LIN {X 0,Y 298.919,Z 282.875,A -85,B 0,C 180,E1 -16201.349,E2 -16201.349} C_VEL
LIN {X 0,Y 298.794,Z 282.889,A -85,B 0,C 180,E1 -16206.755,E2 -16206.755} C_VEL
LIN {X 0,Y 298.677,Z 282.907,A -85,B 0,C 180,E1 -16209.482,E2 -16209.482} C_VEL
LIN {X 0,Y 298.549,Z 282.919,A -85,B 0,C 180,E1 -16213.617,E2 -16213.617} C_VEL
LIN {X 0,Y 298.546,Z 282.921,A -85,B 0,C 180,E1 -16216.41,E2 -16216.41} C_VEL
LIN {X 0,Y 298.509,Z 282.922,A -85,B 0,C 180,E1 -16219.656,E2 -16219.656} C_VEL
LIN {X 0,Y 298.48,Z 283.099,A -85,B 0,C 180,E1 -16223.325,E2 -16223.325} C_VEL
LIN {X 0,Y 298.814,Z 284.83,A -85,B 0,C 180,E1 -16226.655,E2 -16226.655} C_VEL
LIN {X 0,Y 299.125,Z 286.68,A -85,B 0,C 180,E1 -16229.622,E2 -16229.622} C_VEL
LIN {X 0,Y 299.687,Z 290.164,A -85,B 0,C 180,E1 -16234.253,E2 -16234.253} C_VEL
LIN {X 0,Y 300.171,Z 292.989,A -85,B 0,C 180,E1 -16237.5,E2 -16237.5} C_VEL
LIN {X 0,Y 300.838,Z 297.077,A -85,B 0,C 180,E1 -16241.622,E2 -16241.622} C_VEL
LIN {X 0,Y 301.665,Z 301.596,A -85,B 0,C 180,E1 -16245.661,E2 -16245.661} C_VEL
LIN {X 0,Y 301.692,Z 304.757,A -85,B 0,C 180,E1 -16248.199,E2 -16248.199} C_VEL
LIN {X 0,Y 300.821,Z 309.639,A -85,B 0,C 180,E1 -16251.75,E2 -16251.75} C_VEL
LIN {X 0,Y 300.436,Z 312.082,A -85,B 0,C 180,E1 -16253.389,E2 -16253.389} C_VEL
LIN {X 0,Y 301.353,Z 315.27,A -85,B 0,C 180,E1 -16253.65,E2 -16253.65} C_VEL
LIN {X 0,Y 302.505,Z 317.919,A -85,B 0,C 180,E1 -16253.94,E2 -16253.94} C_VEL
LIN {X 0,Y 307.209,Z 331.176,A -85,B 0,C 180,E1 -16255.276,E2 -16255.276} C_VEL
LIN {X 0,Y 310.679,Z 343.941,A -85,B 0,C 180,E1 -16256.565,E2 -16256.565} C_VEL
LIN {X 0,Y 312.999,Z 356.009,A -85,B 0,C 180,E1 -16257.802,E2 -16257.802} C_VEL
LIN {X 0,Y 314.515,Z 369.598,A -85,B 0,C 180,E1 -16259.261,E2 -16259.261} C_VEL
LIN {X 0,Y 315.116,Z 381.128,A -85,B 0,C 180,E1 -16260.617,E2 -16260.617} C_VEL
LIN {X 0,Y 312.318,Z 395,A -85,B 0,C 180,E1 -16262.166,E2 -16262.166} C_VEL
LIN {X 0,Y 309.669,Z 406.556,A -85,B 0,C 180,E1 -16263.734,E2 -16263.734} C_VEL
LIN {X 0,Y 306.844,Z 418.279,A -85,B 0,C 180,E1 -16265.653,E2 -16265.653} C_VEL
LIN {X 0,Y 304.314,Z 429.043,A -85,B 0,C 180,E1 -16267.799,E2 -16267.799} C_VEL
LIN {X 0,Y 302.202,Z 438.027,A -85,B 0,C 180,E1 -16269.94,E2 -16269.94} C_VEL
LIN {X 0,Y 300.309,Z 446.263,A -85,B 0,C 180,E1 -16272.289,E2 -16272.289} C_VEL
LIN {X 0,Y 298.594,Z 453.992,A -85,B 0,C 180,E1 -16274.996,E2 -16274.996} C_VEL
LIN {X 0,Y 297.601,Z 460.201,A -85,B 0,C 180,E1 -16277.73,E2 -16277.73} C_VEL
LIN {X 0,Y 296.971,Z 465.011,A -85,B 0,C 180,E1 -16280.465,E2 -16280.465} C_VEL
LIN {X 0,Y 296.728,Z 468.523,A -85,B 0,C 180,E1 -16283.2,E2 -16283.2} C_VEL
LIN {X 0,Y 296.652,Z 470.817,A -85,B 0,C 180,E1 -16285.925,E2 -16285.925} C_VEL
LIN {X 0,Y 296.663,Z 471.931,A -85,B 0,C 180,E1 -16288.643,E2 -16288.643} C_VEL
LIN {X 0,Y 296.733,Z 472.054,A -85,B 0,C 180,E1 -16290.001,E2 -16290.001} C_VEL
LIN {X 0,Y 296.633,Z 471.4,A -85,B 0,C 180,E1 -16292.717,E2 -16292.717} C_VEL
LIN {X 0,Y 296.692,Z 469.509,A -85,B 0,C 180,E1 -16295.438,E2 -16295.438} C_VEL
LIN {X 0,Y 296.827,Z 466.384,A -85,B 0,C 180,E1 -16298.168,E2 -16298.168} C_VEL
LIN {X 0,Y 297.197,Z 461.97,A -85,B 0,C 180,E1 -16300.906,E2 -16300.906} C_VEL
LIN {X 0,Y 298.046,Z 456.167,A -85,B 0,C 180,E1 -16303.64,E2 -16303.64} C_VEL
LIN {X 0,Y 299.38,Z 448.82,A -85,B 0,C 180,E1 -16306.363,E2 -16306.363} C_VEL
LIN {X 0,Y 300.944,Z 440.958,A -85,B 0,C 180,E1 -16308.731,E2 -16308.731} C_VEL
LIN {X 0,Y 303.074,Z 431.526,A -85,B 0,C 180,E1 -16311.066,E2 -16311.066} C_VEL
LIN {X 0,Y 305.057,Z 421.918,A -85,B 0,C 180,E1 -16313.058,E2 -16313.058} C_VEL
LIN {X 0,Y 307.558,Z 410.541,A -85,B 0,C 180,E1 -16315.009,E2 -16315.009} C_VEL
LIN {X 0,Y 310.005,Z 398.045,A -85,B 0,C 180,E1 -16316.782,E2 -16316.782} C_VEL
LIN {X 0,Y 312.757,Z 384.378,A -85,B 0,C 180,E1 -16318.333,E2 -16318.333} C_VEL
LIN {X 0,Y 313.53,Z 379.839,A -85,B 0,C 180,E1 -16318.782,E2 -16318.782} C_VEL
LIN {X 0,Y 311.965,Z 365.595,A -85,B 0,C 180,E1 -16320.332,E2 -16320.332} C_VEL
LIN {X 0,Y 309.68,Z 351.608,A -85,B 0,C 180,E1 -16321.673,E2 -16321.673} C_VEL
LIN {X 0,Y 306.111,Z 335.839,A -85,B 0,C 180,E1 -16323.017,E2 -16323.017} C_VEL
LIN {X 0,Y 301.772,Z 321.161,A -85,B 0,C 180,E1 -16324.129,E2 -16324.129} C_VEL
LIN {X 0,Y 300.006,Z 315.466,A -85,B 0,C 180,E1 -16324.519,E2 -16324.519} C_VEL
LIN {X 0,Y 299.925,Z 314.804,A -85,B 0,C 180,E1 -16324.578,E2 -16324.578} C_VEL
LIN {X 0,Y 300.788,Z 309.235,A -85,B 0,C 180,E1 -16328.257,E2 -16328.257} C_VEL
LIN {X 0,Y 301.384,Z 305.562,A -85,B 0,C 180,E1 -16330.764,E2 -16330.764} C_VEL
LIN {X 0,Y 301.617,Z 303.07,A -85,B 0,C 180,E1 -16332.512,E2 -16332.512} C_VEL
LIN {X 0,Y 301.57,Z 300.589,A -85,B 0,C 180,E1 -16334.359,E2 -16334.359} C_VEL
LIN {X 0,Y 300.579,Z 295.456,A -85,B 0,C 180,E1 -16338.437,E2 -16338.437} C_VEL
LIN {X 0,Y 299.661,Z 290.232,A -85,B 0,C 180,E1 -16342.884,E2 -16342.884} C_VEL
LIN {X 0,Y 299.197,Z 287.18,A -85,B 0,C 180,E1 -16345.683,E2 -16345.683} C_VEL
LIN {X 0,Y 298.44,Z 283.034,A -85,B 0,C 180,E1 -16349.776,E2 -16349.776} C_VEL
LIN {X 0,Y 298.484,Z 282.93,A -85,B 0,C 180,E1 -16353.476,E2 -16353.476} C_VEL
LIN {X 0,Y 298.442,Z 282.937,A -85,B 0,C 180,E1 -16356.697,E2 -16356.697} C_VEL
LIN {X 0,Y 298.546,Z 282.923,A -85,B 0,C 180,E1 -16360.756,E2 -16360.756} C_VEL
LIN {X 0,Y 298.6,Z 282.916,A -85,B 0,C 180,E1 -16364.994,E2 -16364.994} C_VEL
LIN {X 0,Y 298.597,Z 282.915,A -85,B 0,C 180,E1 -16369.145,E2 -16369.145} C_VEL
LIN {X 0,Y 298.718,Z 282.9,A -85,B 0,C 180,E1 -16371.883,E2 -16371.883} C_VEL
LIN {X 0,Y 298.648,Z 282.911,A -85,B 0,C 180,E1 -16374.597,E2 -16374.597} C_VEL
LIN {X 0,Y 298.928,Z 282.875,A -85,B 0,C 180,E1 -16378.651,E2 -16378.651} C_VEL
LIN {X 0,Y 298.928,Z 282.871,A -85,B 0,C 180,E1 -16381.346,E2 -16381.346} C_VEL
LIN {X 0,Y 298.801,Z 282.889,A -85,B 0,C 180,E1 -16386.752,E2 -16386.752} C_VEL
LIN {X 0,Y 298.684,Z 282.902,A -85,B 0,C 180,E1 -16389.479,E2 -16389.479} C_VEL
LIN {X 0,Y 298.554,Z 282.914,A -85,B 0,C 180,E1 -16393.614,E2 -16393.614} C_VEL
LIN {X 0,Y 298.551,Z 282.921,A -85,B 0,C 180,E1 -16396.407,E2 -16396.407} C_VEL
LIN {X 0,Y 298.513,Z 282.92,A -85,B 0,C 180,E1 -16399.653,E2 -16399.653} C_VEL
LIN {X 0,Y 298.458,Z 282.931,A -85,B 0,C 180,E1 -16403.596,E2 -16403.596} C_VEL
LIN {X 0,Y 298.486,Z 282.924,A -85,B 0,C 180,E1 -16406.573,E2 -16406.573} C_VEL
LIN {X 0,Y 298.416,Z 282.933,A -85,B 0,C 180,E1 -16409.639,E2 -16409.639} C_VEL
LIN {X 0,Y 298.394,Z 282.938,A -85,B 0,C 180,E1 -16412.798,E2 -16412.798} C_VEL
LIN {X 0,Y 298.462,Z 282.926,A -85,B 0,C 180,E1 -16416.81,E2 -16416.81} C_VEL
LIN {X 0,Y 298.411,Z 282.936,A -85,B 0,C 180,E1 -16421.255,E2 -16421.255} C_VEL
LIN {X 0,Y 298.413,Z 282.935,A -85,B 0,C 180,E1 -16425.045,E2 -16425.045} C_VEL
LIN {X 0,Y 298.45,Z 282.927,A -85,B 0,C 180,E1 -16428.748,E2 -16428.748} C_VEL
LIN {X 0,Y 298.442,Z 282.934,A -85,B 0,C 180,E1 -16432.245,E2 -16432.245} C_VEL
LIN {X 0,Y 298.402,Z 282.937,A -85,B 0,C 180,E1 -16435.579,E2 -16435.579} C_VEL
LIN {X 0,Y 298.389,Z 282.94,A -85,B 0,C 180,E1 -16438.79,E2 -16438.79} C_VEL
LIN {X 0,Y 298.469,Z 282.934,A -85,B 0,C 180,E1 -16441.904,E2 -16441.904} C_VEL
LIN {X 0,Y 298.478,Z 282.927,A -85,B 0,C 180,E1 -16444.922,E2 -16444.922} C_VEL
LIN {X 0,Y 298.442,Z 282.934,A -85,B 0,C 180,E1 -16449.314,E2 -16449.314} C_VEL
LIN {X 0,Y 298.529,Z 282.92,A -85,B 0,C 180,E1 -16452.178,E2 -16452.178} C_VEL
LIN {X 0,Y 298.584,Z 282.917,A -85,B 0,C 180,E1 -16454.993,E2 -16454.993} C_VEL
LIN {X 0,Y 298.586,Z 282.916,A -85,B 0,C 180,E1 -16459.145,E2 -16459.145} C_VEL
LIN {X 0,Y 298.748,Z 282.888,A -85,B 0,C 180,E1 -16461.885,E2 -16461.885} C_VEL
LIN {X 0,Y 298.592,Z 282.915,A -85,B 0,C 180,E1 -16464.597,E2 -16464.597} C_VEL
LIN {X 0,Y 298.28,Z 282.958,A -85,B 0,C 180,E1 -16467.298,E2 -16467.298} C_VEL
LIN {X 0,Y 298.703,Z 283.826,A -85,B 0,C 180,E1 -16468.689,E2 -16468.689} C_VEL
LIN {X 0,Y 299.818,Z 287.044,A -85,B 0,C 180,E1 -16468.935,E2 -16468.935} C_VEL
LIN {X 0,Y 305.646,Z 301.861,A -85,B 0,C 180,E1 -16470.26,E2 -16470.26} C_VEL
LIN {X 0,Y 310.151,Z 313.487,A -85,B 0,C 180,E1 -16471.449,E2 -16471.449} C_VEL
LIN {X 0,Y 314.135,Z 327.182,A -85,B 0,C 180,E1 -16472.928,E2 -16472.928} C_VEL
LIN {X 0,Y 315.72,Z 333.801,A -85,B 0,C 180,E1 -16473.69,E2 -16473.69} C_VEL
LIN {X 0,Y 315.258,Z 338.882,A -85,B 0,C 180,E1 -16474.154,E2 -16474.154} C_VEL
LIN {X 0,Y 313.237,Z 352.066,A -85,B 0,C 180,E1 -16475.471,E2 -16475.471} C_VEL
LIN {X 0,Y 311.014,Z 364.333,A -85,B 0,C 180,E1 -16476.958,E2 -16476.958} C_VEL
LIN {X 0,Y 308.798,Z 375.976,A -85,B 0,C 180,E1 -16478.671,E2 -16478.671} C_VEL
LIN {X 0,Y 306.535,Z 386.753,A -85,B 0,C 180,E1 -16480.568,E2 -16480.568} C_VEL
LIN {X 0,Y 304.365,Z 396.697,A -85,B 0,C 180,E1 -16482.671,E2 -16482.671} C_VEL
LIN {X 0,Y 302.151,Z 406.39,A -85,B 0,C 180,E1 -16485.168,E2 -16485.168} C_VEL
LIN {X 0,Y 300.48,Z 414.358,A -85,B 0,C 180,E1 -16487.701,E2 -16487.701} C_VEL
LIN {X 0,Y 299.164,Z 420.286,A -85,B 0,C 180,E1 -16490.008,E2 -16490.008} C_VEL
LIN {X 0,Y 298.31,Z 424.761,A -85,B 0,C 180,E1 -16492.144,E2 -16492.144} C_VEL
LIN {X 0,Y 297.623,Z 428.608,A -85,B 0,C 180,E1 -16494.407,E2 -16494.407} C_VEL
LIN {X 0,Y 297.086,Z 431.545,A -85,B 0,C 180,E1 -16496.709,E2 -16496.709} C_VEL
LIN {X 0,Y 296.755,Z 433.529,A -85,B 0,C 180,E1 -16498.809,E2 -16498.809} C_VEL
LIN {X 0,Y 296.592,Z 434.977,A -85,B 0,C 180,E1 -16501.459,E2 -16501.459} C_VEL
LIN {X 0,Y 296.562,Z 435.382,A -85,B 0,C 180,E1 -16503.963,E2 -16503.963} C_VEL
LIN {X 0,Y 296.697,Z 434.896,A -85,B 0,C 180,E1 -16506.357,E2 -16506.357} C_VEL
LIN {X 0,Y 297.054,Z 433.533,A -85,B 0,C 180,E1 -16508.674,E2 -16508.674} C_VEL
LIN {X 0,Y 297.695,Z 430.916,A -85,B 0,C 180,E1 -16511.377,E2 -16511.377} C_VEL
LIN {X 0,Y 298.593,Z 427.274,A -85,B 0,C 180,E1 -16513.973,E2 -16513.973} C_VEL
LIN {X 0,Y 299.829,Z 422.32,A -85,B 0,C 180,E1 -16516.604,E2 -16516.604} C_VEL
LIN {X 0,Y 301.488,Z 415.919,A -85,B 0,C 180,E1 -16519.256,E2 -16519.256} C_VEL
LIN {X 0,Y 303.672,Z 407.901,A -85,B 0,C 180,E1 -16521.893,E2 -16521.893} C_VEL
LIN {X 0,Y 305.787,Z 399.629,A -85,B 0,C 180,E1 -16524.11,E2 -16524.11} C_VEL
LIN {X 0,Y 308.375,Z 389.763,A -85,B 0,C 180,E1 -16526.288,E2 -16526.288} C_VEL
LIN {X 0,Y 310.943,Z 379.241,A -85,B 0,C 180,E1 -16528.217,E2 -16528.217} C_VEL
LIN {X 0,Y 313.577,Z 367.883,A -85,B 0,C 180,E1 -16529.94,E2 -16529.94} C_VEL
LIN {X 0,Y 316.01,Z 355.888,A -85,B 0,C 180,E1 -16531.456,E2 -16531.456} C_VEL
LIN {X 0,Y 318.371,Z 343.09,A -85,B 0,C 180,E1 -16532.775,E2 -16532.775} C_VEL
LIN {X 0,Y 319.093,Z 338.798,A -85,B 0,C 180,E1 -16533.161,E2 -16533.161} C_VEL
LIN {X 0,Y 316.264,Z 327.369,A -85,B 0,C 180,E1 -16534.642,E2 -16534.642} C_VEL
LIN {X 0,Y 311.737,Z 314.131,A -85,B 0,C 180,E1 -16536.338,E2 -16536.338} C_VEL
LIN {X 0,Y 306.157,Z 301.839,A -85,B 0,C 180,E1 -16537.966,E2 -16537.966} C_VEL
LIN {X 0,Y 302.671,Z 295.179,A -85,B 0,C 180,E1 -16538.863,E2 -16538.863} C_VEL
LIN {X 0,Y 300.761,Z 291.735,A -85,B 0,C 180,E1 -16539.323,E2 -16539.323} C_VEL
LIN {X 0,Y 299.162,Z 288.982,A -85,B 0,C 180,E1 -16539.713,E2 -16539.713} C_VEL
LIN {X 0,Y 298.817,Z 287.666,A -85,B 0,C 180,E1 -16539.845,E2 -16539.845} C_VEL
LIN {X 0,Y 298.868,Z 287.057,A -85,B 0,C 180,E1 -16541.023,E2 -16541.023} C_VEL
LIN {X 0,Y 298.189,Z 286.627,A -85,B 0,C 180,E1 -16542.146,E2 -16542.146} C_VEL
LIN {X 0,Y 295.347,Z 286.279,A -85,B 0,C 180,E1 -16543.98,E2 -16543.98} C_VEL
LIN {X 0,Y 292.934,Z 286.066,A -85,B 0,C 180,E1 -16545.468,E2 -16545.468} C_VEL
LIN {X 0,Y 291.882,Z 285.781,A -85,B 0,C 180,E1 -16546.62,E2 -16546.62} C_VEL
LIN {X 0,Y 291.786,Z 285.628,A -85,B 0,C 180,E1 -16547.009,E2 -16547.009} C_VEL
LIN {X 0,Y 291.735,Z 283.882,A -85,B 0,C 180,E1 -16551.691,E2 -16551.691} C_VEL
LIN {X 0,Y 291.627,Z 283.783,A -85,B 0,C 180,E1 -16554.47,E2 -16554.47} C_VEL
LIN {X 0,Y 291.885,Z 283.752,A -85,B 0,C 180,E1 -16558.622,E2 -16558.622} C_VEL
LIN {X 0,Y 291.886,Z 283.75,A -85,B 0,C 180,E1 -16561.381,E2 -16561.381} C_VEL
LIN {X 0,Y 291.743,Z 283.768,A -85,B 0,C 180,E1 -16566.919,E2 -16566.919} C_VEL
LIN {X 0,Y 291.626,Z 283.785,A -85,B 0,C 180,E1 -16569.713,E2 -16569.713} C_VEL
LIN {X 0,Y 291.519,Z 283.797,A -85,B 0,C 180,E1 -16573.952,E2 -16573.952} C_VEL
LIN {X 0,Y 291.484,Z 283.797,A -85,B 0,C 180,E1 -16576.819,E2 -16576.819} C_VEL
LIN {X 0,Y 291.448,Z 283.803,A -85,B 0,C 180,E1 -16579.876,E2 -16579.876} C_VEL
LIN {X 0,Y 291.396,Z 283.873,A -85,B 0,C 180,E1 -16581.211,E2 -16581.211} C_VEL
LIN {X 0,Y 291.623,Z 285.187,A -85,B 0,C 180,E1 -16584.187,E2 -16584.187} C_VEL
LIN {X 0,Y 291.966,Z 286.805,A -85,B 0,C 180,E1 -16587.218,E2 -16587.218} C_VEL
LIN {X 0,Y 292.243,Z 288.784,A -85,B 0,C 180,E1 -16590.334,E2 -16590.334} C_VEL
LIN {X 0,Y 292.62,Z 291.137,A -85,B 0,C 180,E1 -16593.533,E2 -16593.533} C_VEL
LIN {X 0,Y 293.13,Z 293.884,A -85,B 0,C 180,E1 -16596.828,E2 -16596.828} C_VEL
LIN {X 0,Y 293.626,Z 297.12,A -85,B 0,C 180,E1 -16600.261,E2 -16600.261} C_VEL
LIN {X 0,Y 294.415,Z 301.316,A -85,B 0,C 180,E1 -16604.265,E2 -16604.265} C_VEL
LIN {X 0,Y 294.753,Z 303.579,A -85,B 0,C 180,E1 -16606.255,E2 -16606.255} C_VEL
LIN {X 0,Y 294.711,Z 305.868,A -85,B 0,C 180,E1 -16608.11,E2 -16608.11} C_VEL
LIN {X 0,Y 293.689,Z 311.336,A -85,B 0,C 180,E1 -16612.185,E2 -16612.185} C_VEL
LIN {X 0,Y 294.665,Z 314.757,A -85,B 0,C 180,E1 -16612.509,E2 -16612.509} C_VEL
LIN {X 0,Y 295.761,Z 317.224,A -85,B 0,C 180,E1 -16612.804,E2 -16612.804} C_VEL
LIN {X 0,Y 300.269,Z 329.416,A -85,B 0,C 180,E1 -16614.128,E2 -16614.128} C_VEL
LIN {X 0,Y 304.198,Z 343.339,A -85,B 0,C 180,E1 -16615.627,E2 -16615.627} C_VEL
LIN {X 0,Y 306.889,Z 357.513,A -85,B 0,C 180,E1 -16617.159,E2 -16617.159} C_VEL
LIN {X 0,Y 308.218,Z 370.175,A -85,B 0,C 180,E1 -16618.584,E2 -16618.584} C_VEL
LIN {X 0,Y 308.727,Z 382.548,A -85,B 0,C 180,E1 -16620.097,E2 -16620.097} C_VEL
LIN {X 0,Y 305.76,Z 396.324,A -85,B 0,C 180,E1 -16621.702,E2 -16621.702} C_VEL
LIN {X 0,Y 302.793,Z 408.654,A -85,B 0,C 180,E1 -16623.462,E2 -16623.462} C_VEL
LIN {X 0,Y 299.919,Z 419.961,A -85,B 0,C 180,E1 -16625.423,E2 -16625.423} C_VEL
LIN {X 0,Y 297.23,Z 431.049,A -85,B 0,C 180,E1 -16627.771,E2 -16627.771} C_VEL
LIN {X 0,Y 294.831,Z 440.289,A -85,B 0,C 180,E1 -16630.144,E2 -16630.144} C_VEL
LIN {X 0,Y 293.012,Z 448.031,A -85,B 0,C 180,E1 -16632.554,E2 -16632.554} C_VEL
LIN {X 0,Y 291.352,Z 455.328,A -85,B 0,C 180,E1 -16635.329,E2 -16635.329} C_VEL
LIN {X 0,Y 290.374,Z 461.138,A -85,B 0,C 180,E1 -16638.129,E2 -16638.129} C_VEL
LIN {X 0,Y 289.911,Z 464.645,A -85,B 0,C 180,E1 -16640.231,E2 -16640.231} C_VEL
LIN {X 0,Y 289.649,Z 468.132,A -85,B 0,C 180,E1 -16643.033,E2 -16643.033} C_VEL
LIN {X 0,Y 289.57,Z 470.402,A -85,B 0,C 180,E1 -16645.825,E2 -16645.825} C_VEL
LIN {X 0,Y 289.575,Z 471.496,A -85,B 0,C 180,E1 -16648.61,E2 -16648.61} C_VEL
LIN {X 0,Y 289.646,Z 471.609,A -85,B 0,C 180,E1 -16650.001,E2 -16650.001} C_VEL
LIN {X 0,Y 289.558,Z 470.938,A -85,B 0,C 180,E1 -16652.783,E2 -16652.783} C_VEL
LIN {X 0,Y 289.642,Z 468.827,A -85,B 0,C 180,E1 -16655.814,E2 -16655.814} C_VEL
LIN {X 0,Y 289.837,Z 464.915,A -85,B 0,C 180,E1 -16659.069,E2 -16659.069} C_VEL
LIN {X 0,Y 290.376,Z 460.158,A -85,B 0,C 180,E1 -16661.873,E2 -16661.873} C_VEL
LIN {X 0,Y 291.365,Z 453.952,A -85,B 0,C 180,E1 -16664.672,E2 -16664.672} C_VEL
LIN {X 0,Y 292.919,Z 446.146,A -85,B 0,C 180,E1 -16667.453,E2 -16667.453} C_VEL
LIN {X 0,Y 294.737,Z 437.817,A -85,B 0,C 180,E1 -16669.865,E2 -16669.865} C_VEL
LIN {X 0,Y 297.028,Z 427.814,A -85,B 0,C 180,E1 -16672.247,E2 -16672.247} C_VEL
LIN {X 0,Y 299.237,Z 417.559,A -85,B 0,C 180,E1 -16674.269,E2 -16674.269} C_VEL
LIN {X 0,Y 301.992,Z 405.418,A -85,B 0,C 180,E1 -16676.243,E2 -16676.243} C_VEL
LIN {X 0,Y 304.194,Z 394.565,A -85,B 0,C 180,E1 -16677.709,E2 -16677.709} C_VEL
LIN {X 0,Y 306.655,Z 382.432,A -85,B 0,C 180,E1 -16679.063,E2 -16679.063} C_VEL
LIN {X 0,Y 306.745,Z 378.889,A -85,B 0,C 180,E1 -16679.465,E2 -16679.465} C_VEL
LIN {X 0,Y 305.283,Z 365.72,A -85,B 0,C 180,E1 -16680.941,E2 -16680.941} C_VEL
LIN {X 0,Y 303.087,Z 352,A -85,B 0,C 180,E1 -16682.307,E2 -16682.307} C_VEL
LIN {X 0,Y 299.567,Z 336.367,A -85,B 0,C 180,E1 -16683.689,E2 -16683.689} C_VEL
LIN {X 0,Y 294.917,Z 320.751,A -85,B 0,C 180,E1 -16684.933,E2 -16684.933} C_VEL
LIN {X 0,Y 293.131,Z 315.095,A -85,B 0,C 180,E1 -16685.343,E2 -16685.343} C_VEL
LIN {X 0,Y 293.075,Z 314.35,A -85,B 0,C 180,E1 -16685.404,E2 -16685.404} C_VEL
LIN {X 0,Y 294.007,Z 308.671,A -85,B 0,C 180,E1 -16689.297,E2 -16689.297} C_VEL
LIN {X 0,Y 294.587,Z 304.45,A -85,B 0,C 180,E1 -16692.304,E2 -16692.304} C_VEL
LIN {X 0,Y 294.564,Z 301.822,A -85,B 0,C 180,E1 -16694.292,E2 -16694.292} C_VEL
LIN {X 0,Y 293.684,Z 297.304,A -85,B 0,C 180,E1 -16697.927,E2 -16697.927} C_VEL
LIN {X 0,Y 292.948,Z 293.24,A -85,B 0,C 180,E1 -16701.408,E2 -16701.408} C_VEL
LIN {X 0,Y 292.364,Z 289.487,A -85,B 0,C 180,E1 -16704.818,E2 -16704.818} C_VEL
LIN {X 0,Y 291.818,Z 286.231,A -85,B 0,C 180,E1 -16708.004,E2 -16708.004} C_VEL
LIN {X 0,Y 291.404,Z 283.813,A -85,B 0,C 180,E1 -16710.704,E2 -16710.704} C_VEL
LIN {X 0,Y 291.419,Z 283.811,A -85,B 0,C 180,E1 -16714.271,E2 -16714.271} C_VEL
LIN {X 0,Y 291.388,Z 283.814,A -85,B 0,C 180,E1 -16717.299,E2 -16717.299} C_VEL
LIN {X 0,Y 291.464,Z 283.805,A -85,B 0,C 180,E1 -16720.269,E2 -16720.269} C_VEL
LIN {X 0,Y 291.561,Z 283.795,A -85,B 0,C 180,E1 -16724.623,E2 -16724.623} C_VEL
LIN {X 0,Y 291.541,Z 283.796,A -85,B 0,C 180,E1 -16728.879,E2 -16728.879} C_VEL
LIN {X 0,Y 291.669,Z 283.778,A -85,B 0,C 180,E1 -16731.686,E2 -16731.686} C_VEL
LIN {X 0,Y 291.617,Z 283.788,A -85,B 0,C 180,E1 -16734.467,E2 -16734.467} C_VEL
LIN {X 0,Y 291.894,Z 283.752,A -85,B 0,C 180,E1 -16738.619,E2 -16738.619} C_VEL
LIN {X 0,Y 291.894,Z 283.748,A -85,B 0,C 180,E1 -16741.378,E2 -16741.378} C_VEL
LIN {X 0,Y 291.75,Z 283.766,A -85,B 0,C 180,E1 -16746.916,E2 -16746.916} C_VEL
LIN {X 0,Y 291.633,Z 283.781,A -85,B 0,C 180,E1 -16749.71,E2 -16749.71} C_VEL
LIN {X 0,Y 291.524,Z 283.791,A -85,B 0,C 180,E1 -16753.948,E2 -16753.948} C_VEL
LIN {X 0,Y 291.489,Z 283.798,A -85,B 0,C 180,E1 -16756.816,E2 -16756.816} C_VEL
LIN {X 0,Y 291.452,Z 283.799,A -85,B 0,C 180,E1 -16759.873,E2 -16759.873} C_VEL
LIN {X 0,Y 291.401,Z 283.813,A -85,B 0,C 180,E1 -16764.203,E2 -16764.203} C_VEL
LIN {X 0,Y 291.419,Z 283.803,A -85,B 0,C 180,E1 -16767.27,E2 -16767.27} C_VEL
LIN {X 0,Y 291.333,Z 283.819,A -85,B 0,C 180,E1 -16770.435,E2 -16770.435} C_VEL
LIN {X 0,Y 291.343,Z 283.819,A -85,B 0,C 180,E1 -16773.696,E2 -16773.696} C_VEL
LIN {X 0,Y 291.391,Z 283.807,A -85,B 0,C 180,E1 -16777.256,E2 -16777.256} C_VEL
LIN {X 0,Y 291.368,Z 283.813,A -85,B 0,C 180,E1 -16780.634,E2 -16780.634} C_VEL
LIN {X 0,Y 291.339,Z 283.817,A -85,B 0,C 180,E1 -16784.39,E2 -16784.39} C_VEL
LIN {X 0,Y 291.384,Z 283.808,A -85,B 0,C 180,E1 -16788.388,E2 -16788.388} C_VEL
LIN {X 0,Y 291.383,Z 283.811,A -85,B 0,C 180,E1 -16791.162,E2 -16791.162} C_VEL
LIN {X 0,Y 291.38,Z 283.808,A -85,B 0,C 180,E1 -16794.628,E2 -16794.628} C_VEL
LIN {X 0,Y 291.366,Z 283.817,A -85,B 0,C 180,E1 -16797.949,E2 -16797.949} C_VEL
LIN {X 0,Y 291.383,Z 283.812,A -85,B 0,C 180,E1 -16801.157,E2 -16801.157} C_VEL
LIN {X 0,Y 291.414,Z 283.807,A -85,B 0,C 180,E1 -16804.271,E2 -16804.271} C_VEL
LIN {X 0,Y 291.374,Z 283.818,A -85,B 0,C 180,E1 -16807.298,E2 -16807.298} C_VEL
LIN {X 0,Y 291.45,Z 283.805,A -85,B 0,C 180,E1 -16810.269,E2 -16810.269} C_VEL
LIN {X 0,Y 291.547,Z 283.792,A -85,B 0,C 180,E1 -16814.622,E2 -16814.622} C_VEL
LIN {X 0,Y 291.529,Z 283.794,A -85,B 0,C 180,E1 -16818.879,E2 -16818.879} C_VEL
LIN {X 0,Y 291.698,Z 283.767,A -85,B 0,C 180,E1 -16821.687,E2 -16821.687} C_VEL
LIN {X 0,Y 291.57,Z 283.79,A -85,B 0,C 180,E1 -16824.466,E2 -16824.466} C_VEL
LIN {X 0,Y 291.239,Z 283.892,A -85,B 0,C 180,E1 -16827.233,E2 -16827.233} C_VEL
LIN {X 0,Y 291.409,Z 284.249,A -85,B 0,C 180,E1 -16827.805,E2 -16827.805} C_VEL
LIN {X 0,Y 292.558,Z 287.296,A -85,B 0,C 180,E1 -16828.063,E2 -16828.063} C_VEL
LIN {X 0,Y 293.711,Z 289.342,A -85,B 0,C 180,E1 -16828.281,E2 -16828.281} C_VEL
LIN {X 0,Y 299.354,Z 303.678,A -85,B 0,C 180,E1 -16829.642,E2 -16829.642} C_VEL
LIN {X 0,Y 304.299,Z 317.05,A -85,B 0,C 180,E1 -16831.079,E2 -16831.079} C_VEL
LIN {X 0,Y 308.101,Z 330.596,A -85,B 0,C 180,E1 -16832.614,E2 -16832.614} C_VEL
LIN {X 0,Y 309.356,Z 335.929,A -85,B 0,C 180,E1 -16833.255,E2 -16833.255} C_VEL
LIN {X 0,Y 307.295,Z 349.677,A -85,B 0,C 180,E1 -16834.59,E2 -16834.59} C_VEL
LIN {X 0,Y 305.023,Z 362.473,A -85,B 0,C 180,E1 -16836.116,E2 -16836.116} C_VEL
LIN {X 0,Y 302.438,Z 375.466,A -85,B 0,C 180,E1 -16838.014,E2 -16838.014} C_VEL
LIN {X 0,Y 299.846,Z 387.337,A -85,B 0,C 180,E1 -16840.138,E2 -16840.138} C_VEL
LIN {X 0,Y 297.596,Z 397.206,A -85,B 0,C 180,E1 -16842.27,E2 -16842.27} C_VEL
LIN {X 0,Y 295.319,Z 406.878,A -85,B 0,C 180,E1 -16844.822,E2 -16844.822} C_VEL
LIN {X 0,Y 293.525,Z 415.004,A -85,B 0,C 180,E1 -16847.473,E2 -16847.473} C_VEL
LIN {X 0,Y 292.003,Z 421.677,A -85,B 0,C 180,E1 -16850.178,E2 -16850.178} C_VEL
LIN {X 0,Y 290.842,Z 427.612,A -85,B 0,C 180,E1 -16853.335,E2 -16853.335} C_VEL
LIN {X 0,Y 290.102,Z 431.671,A -85,B 0,C 180,E1 -16856.321,E2 -16856.321} C_VEL
LIN {X 0,Y 289.626,Z 434.228,A -85,B 0,C 180,E1 -16859.128,E2 -16859.128} C_VEL
LIN {X 0,Y 289.47,Z 435.667,A -85,B 0,C 180,E1 -16862.284,E2 -16862.284} C_VEL
LIN {X 0,Y 289.507,Z 435.805,A -85,B 0,C 180,E1 -16864.377,E2 -16864.377} C_VEL
LIN {X 0,Y 289.717,Z 434.943,A -85,B 0,C 180,E1 -16867.332,E2 -16867.332} C_VEL
LIN {X 0,Y 290.06,Z 433.761,A -85,B 0,C 180,E1 -16869.167,E2 -16869.167} C_VEL
LIN {X 0,Y 290.648,Z 431.602,A -85,B 0,C 180,E1 -16871.448,E2 -16871.448} C_VEL
LIN {X 0,Y 291.673,Z 427.685,A -85,B 0,C 180,E1 -16874.327,E2 -16874.327} C_VEL
LIN {X 0,Y 292.996,Z 422.745,A -85,B 0,C 180,E1 -16877.008,E2 -16877.008} C_VEL
LIN {X 0,Y 294.956,Z 415.697,A -85,B 0,C 180,E1 -16879.961,E2 -16879.961} C_VEL
LIN {X 0,Y 297.229,Z 407.744,A -85,B 0,C 180,E1 -16882.58,E2 -16882.58} C_VEL
LIN {X 0,Y 299.796,Z 398.182,A -85,B 0,C 180,E1 -16885.132,E2 -16885.132} C_VEL
LIN {X 0,Y 302.573,Z 387.97,A -85,B 0,C 180,E1 -16887.344,E2 -16887.344} C_VEL
LIN {X 0,Y 305.563,Z 376.305,A -85,B 0,C 180,E1 -16889.407,E2 -16889.407} C_VEL
LIN {X 0,Y 308.354,Z 364.087,A -85,B 0,C 180,E1 -16891.185,E2 -16891.185} C_VEL
LIN {X 0,Y 311.059,Z 351.004,A -85,B 0,C 180,E1 -16892.733,E2 -16892.733} C_VEL
LIN {X 0,Y 312.951,Z 340.409,A -85,B 0,C 180,E1 -16893.772,E2 -16893.772} C_VEL
LIN {X 0,Y 309.972,Z 328.735,A -85,B 0,C 180,E1 -16895.381,E2 -16895.381} C_VEL
LIN {X 0,Y 305.839,Z 316.513,A -85,B 0,C 180,E1 -16897.04,E2 -16897.04} C_VEL
LIN {X 0,Y 300.303,Z 304.008,A -85,B 0,C 180,E1 -16898.778,E2 -16898.778} C_VEL
LIN {X 0,Y 295.805,Z 295.796,A -85,B 0,C 180,E1 -16900.004,E2 -16900.004} C_VEL
LIN {X 0,Y 293.912,Z 292.439,A -85,B 0,C 180,E1 -16900.489,E2 -16900.489} C_VEL
LIN {X 0,Y 292.239,Z 289.598,A -85,B 0,C 180,E1 -16900.92,E2 -16900.92} C_VEL
LIN {X 0,Y 291.89,Z 288.279,A -85,B 0,C 180,E1 -16901.079,E2 -16901.079} C_VEL
LIN {X 0,Y 291.945,Z 286.613,A -85,B 0,C 180,E1 -16904.646,E2 -16904.646} C_VEL
LIN {X 0,Y 291.786,Z 285.628,A -85,B 0,C 180,E1 -16907.009,E2 -16907.009} C_VEL
LIN {X 0,Y 291.113,Z 285.308,A -85,B 0,C 180,E1 -16908.16,E2 -16908.16} C_VEL
LIN {X 0,Y 288.329,Z 285.148,A -85,B 0,C 180,E1 -16910.04,E2 -16910.04} C_VEL
LIN {X 0,Y 285.09,Z 285.041,A -85,B 0,C 180,E1 -16912.349,E2 -16912.349} C_VEL
LIN {X 0,Y 284.7,Z 284.892,A -85,B 0,C 180,E1 -16913.146,E2 -16913.146} C_VEL
LIN {X 0,Y 284.851,Z 284.628,A -85,B 0,C 180,E1 -16918.588,E2 -16918.588} C_VEL
LIN {X 0,Y 284.852,Z 284.626,A -85,B 0,C 180,E1 -16921.415,E2 -16921.415} C_VEL
LIN {X 0,Y 284.695,Z 284.647,A -85,B 0,C 180,E1 -16927.092,E2 -16927.092} C_VEL
LIN {X 0,Y 284.563,Z 284.662,A -85,B 0,C 180,E1 -16929.957,E2 -16929.957} C_VEL
LIN {X 0,Y 284.478,Z 284.672,A -85,B 0,C 180,E1 -16934.304,E2 -16934.304} C_VEL
LIN {X 0,Y 284.423,Z 284.676,A -85,B 0,C 180,E1 -16937.25,E2 -16937.25} C_VEL
LIN {X 0,Y 284.402,Z 284.681,A -85,B 0,C 180,E1 -16938.74,E2 -16938.74} C_VEL
LIN {X 0,Y 284.51,Z 285.77,A -85,B 0,C 180,E1 -16941.75,E2 -16941.75} C_VEL
LIN {X 0,Y 284.775,Z 287.16,A -85,B 0,C 180,E1 -16944.807,E2 -16944.807} C_VEL
LIN {X 0,Y 285.111,Z 288.859,A -85,B 0,C 180,E1 -16947.929,E2 -16947.929} C_VEL
LIN {X 0,Y 285.397,Z 290.95,A -85,B 0,C 180,E1 -16951.141,E2 -16951.141} C_VEL
LIN {X 0,Y 285.82,Z 293.416,A -85,B 0,C 180,E1 -16954.441,E2 -16954.441} C_VEL
LIN {X 0,Y 286.377,Z 296.662,A -85,B 0,C 180,E1 -16958.252,E2 -16958.252} C_VEL
LIN {X 0,Y 287.089,Z 301.038,A -85,B 0,C 180,E1 -16962.745,E2 -16962.745} C_VEL
LIN {X 0,Y 287.602,Z 303.585,A -85,B 0,C 180,E1 -16965.127,E2 -16965.127} C_VEL
LIN {X 0,Y 287.775,Z 305.866,A -85,B 0,C 180,E1 -16967.111,E2 -16967.111} C_VEL
LIN {X 0,Y 287.394,Z 308.614,A -85,B 0,C 180,E1 -16969.297,E2 -16969.297} C_VEL
LIN {X 0,Y 286.973,Z 310.742,A -85,B 0,C 180,E1 -16970.935,E2 -16970.935} C_VEL
LIN {X 0,Y 287.896,Z 314.026,A -85,B 0,C 180,E1 -16971.254,E2 -16971.254} C_VEL
LIN {X 0,Y 289.163,Z 316.7,A -85,B 0,C 180,E1 -16971.607,E2 -16971.607} C_VEL
LIN {X 0,Y 293.899,Z 329.427,A -85,B 0,C 180,E1 -16973.093,E2 -16973.093} C_VEL
LIN {X 0,Y 297.914,Z 343.493,A -85,B 0,C 180,E1 -16974.706,E2 -16974.706} C_VEL
LIN {X 0,Y 300.394,Z 356.178,A -85,B 0,C 180,E1 -16976.156,E2 -16976.156} C_VEL
LIN {X 0,Y 301.828,Z 368.687,A -85,B 0,C 180,E1 -16977.62,E2 -16977.62} C_VEL
LIN {X 0,Y 302.357,Z 382.227,A -85,B 0,C 180,E1 -16979.321,E2 -16979.321} C_VEL
LIN {X 0,Y 302.01,Z 385.661,A -85,B 0,C 180,E1 -16979.753,E2 -16979.753} C_VEL
LIN {X 0,Y 298.921,Z 398.741,A -85,B 0,C 180,E1 -16981.378,E2 -16981.378} C_VEL
LIN {X 0,Y 295.857,Z 410.581,A -85,B 0,C 180,E1 -16983.171,E2 -16983.171} C_VEL
LIN {X 0,Y 292.976,Z 421.521,A -85,B 0,C 180,E1 -16985.179,E2 -16985.179} C_VEL
LIN {X 0,Y 290.567,Z 430.873,A -85,B 0,C 180,E1 -16987.233,E2 -16987.233} C_VEL
LIN {X 0,Y 288.106,Z 440.075,A -85,B 0,C 180,E1 -16989.66,E2 -16989.66} C_VEL
LIN {X 0,Y 286.151,Z 447.768,A -85,B 0,C 180,E1 -16992.122,E2 -16992.122} C_VEL
LIN {X 0,Y 284.401,Z 455.06,A -85,B 0,C 180,E1 -16994.983,E2 -16994.983} C_VEL
LIN {X 0,Y 283.359,Z 460.785,A -85,B 0,C 180,E1 -16997.831,E2 -16997.831} C_VEL
LIN {X 0,Y 282.842,Z 464.274,A -85,B 0,C 180,E1 -16999.984,E2 -16999.984} C_VEL
LIN {X 0,Y 282.571,Z 467.745,A -85,B 0,C 180,E1 -17002.857,E2 -17002.857} C_VEL
LIN {X 0,Y 282.492,Z 469.991,A -85,B 0,C 180,E1 -17005.721,E2 -17005.721} C_VEL
LIN {X 0,Y 282.491,Z 471.061,A -85,B 0,C 180,E1 -17008.575,E2 -17008.575} C_VEL
LIN {X 0,Y 282.559,Z 471.161,A -85,B 0,C 180,E1 -17010.001,E2 -17010.001} C_VEL
LIN {X 0,Y 282.485,Z 470.466,A -85,B 0,C 180,E1 -17012.853,E2 -17012.853} C_VEL
LIN {X 0,Y 282.562,Z 468.491,A -85,B 0,C 180,E1 -17015.783,E2 -17015.783} C_VEL
LIN {X 0,Y 282.699,Z 465.368,A -85,B 0,C 180,E1 -17018.579,E2 -17018.579} C_VEL
LIN {X 0,Y 283.136,Z 460.893,A -85,B 0,C 180,E1 -17021.455,E2 -17021.455} C_VEL
LIN {X 0,Y 284.11,Z 455.022,A -85,B 0,C 180,E1 -17024.323,E2 -17024.323} C_VEL
LIN {X 0,Y 285.595,Z 447.599,A -85,B 0,C 180,E1 -17027.176,E2 -17027.176} C_VEL
LIN {X 0,Y 287.317,Z 439.648,A -85,B 0,C 180,E1 -17029.655,E2 -17029.655} C_VEL
LIN {X 0,Y 289.627,Z 430.114,A -85,B 0,C 180,E1 -17032.094,E2 -17032.094} C_VEL
LIN {X 0,Y 291.857,Z 420.399,A -85,B 0,C 180,E1 -17034.166,E2 -17034.166} C_VEL
LIN {X 0,Y 294.569,Z 408.896,A -85,B 0,C 180,E1 -17036.193,E2 -17036.193} C_VEL
LIN {X 0,Y 297.289,Z 396.253,A -85,B 0,C 180,E1 -17038.026,E2 -17038.026} C_VEL
LIN {X 0,Y 300.059,Z 383.292,A -85,B 0,C 180,E1 -17039.538,E2 -17039.538} C_VEL
LIN {X 0,Y 300.117,Z 379.784,A -85,B 0,C 180,E1 -17039.95,E2 -17039.95} C_VEL
LIN {X 0,Y 298.622,Z 365.497,A -85,B 0,C 180,E1 -17041.606,E2 -17041.606} C_VEL
LIN {X 0,Y 296.219,Z 351.264,A -85,B 0,C 180,E1 -17043.073,E2 -17043.073} C_VEL
LIN {X 0,Y 292.731,Z 335.733,A -85,B 0,C 180,E1 -17044.493,E2 -17044.493} C_VEL
LIN {X 0,Y 288.206,Z 320.737,A -85,B 0,C 180,E1 -17045.75,E2 -17045.75} C_VEL
LIN {X 0,Y 286.285,Z 314.556,A -85,B 0,C 180,E1 -17046.209,E2 -17046.209} C_VEL
LIN {X 0,Y 286.223,Z 313.881,A -85,B 0,C 180,E1 -17046.305,E2 -17046.305} C_VEL
LIN {X 0,Y 287.286,Z 307.716,A -85,B 0,C 180,E1 -17050.678,E2 -17050.678} C_VEL
LIN {X 0,Y 287.564,Z 304.367,A -85,B 0,C 180,E1 -17053.183,E2 -17053.183} C_VEL
LIN {X 0,Y 287.338,Z 301.821,A -85,B 0,C 180,E1 -17055.18,E2 -17055.18} C_VEL
LIN {X 0,Y 286.573,Z 297.805,A -85,B 0,C 180,E1 -17058.534,E2 -17058.534} C_VEL
LIN {X 0,Y 285.84,Z 293.807,A -85,B 0,C 180,E1 -17062.07,E2 -17062.07} C_VEL
LIN {X 0,Y 285.263,Z 290.187,A -85,B 0,C 180,E1 -17065.482,E2 -17065.482} C_VEL
LIN {X 0,Y 284.719,Z 286.924,A -85,B 0,C 180,E1 -17068.776,E2 -17068.776} C_VEL
LIN {X 0,Y 284.34,Z 284.694,A -85,B 0,C 180,E1 -17071.184,E2 -17071.184} C_VEL
LIN {X 0,Y 284.381,Z 284.688,A -85,B 0,C 180,E1 -17073.586,E2 -17073.586} C_VEL
LIN {X 0,Y 284.373,Z 284.689,A -85,B 0,C 180,E1 -17076.706,E2 -17076.706} C_VEL
LIN {X 0,Y 284.41,Z 284.682,A -85,B 0,C 180,E1 -17081.261,E2 -17081.261} C_VEL
LIN {X 0,Y 284.498,Z 284.675,A -85,B 0,C 180,E1 -17084.458,E2 -17084.458} C_VEL
LIN {X 0,Y 284.493,Z 284.676,A -85,B 0,C 180,E1 -17088.6,E2 -17088.6} C_VEL
LIN {X 0,Y 284.624,Z 284.656,A -85,B 0,C 180,E1 -17091.479,E2 -17091.479} C_VEL
LIN {X 0,Y 284.586,Z 284.663,A -85,B 0,C 180,E1 -17094.33,E2 -17094.33} C_VEL
LIN {X 0,Y 284.86,Z 284.628,A -85,B 0,C 180,E1 -17098.585,E2 -17098.585} C_VEL
LIN {X 0,Y 284.86,Z 284.624,A -85,B 0,C 180,E1 -17101.412,E2 -17101.412} C_VEL
LIN {X 0,Y 284.702,Z 284.643,A -85,B 0,C 180,E1 -17107.088,E2 -17107.088} C_VEL
LIN {X 0,Y 284.57,Z 284.662,A -85,B 0,C 180,E1 -17109.954,E2 -17109.954} C_VEL
LIN {X 0,Y 284.484,Z 284.671,A -85,B 0,C 180,E1 -17114.301,E2 -17114.301} C_VEL
LIN {X 0,Y 284.427,Z 284.677,A -85,B 0,C 180,E1 -17117.246,E2 -17117.246} C_VEL
LIN {X 0,Y 284.38,Z 284.678,A -85,B 0,C 180,E1 -17120.24,E2 -17120.24} C_VEL
LIN {X 0,Y 284.37,Z 284.688,A -85,B 0,C 180,E1 -17123.873,E2 -17123.873} C_VEL
LIN {X 0,Y 284.395,Z 284.677,A -85,B 0,C 180,E1 -17127.171,E2 -17127.171} C_VEL
LIN {X 0,Y 284.293,Z 284.695,A -85,B 0,C 180,E1 -17131.272,E2 -17131.272} C_VEL
LIN {X 0,Y 284.36,Z 284.682,A -85,B 0,C 180,E1 -17135.352,E2 -17135.352} C_VEL
LIN {X 0,Y 284.32,Z 284.694,A -85,B 0,C 180,E1 -17138.165,E2 -17138.165} C_VEL
LIN {X 0,Y 284.293,Z 284.689,A -85,B 0,C 180,E1 -17142.129,E2 -17142.129} C_VEL
LIN {X 0,Y 284.314,Z 284.694,A -85,B 0,C 180,E1 -17146.199,E2 -17146.199} C_VEL
LIN {X 0,Y 284.347,Z 284.687,A -85,B 0,C 180,E1 -17150.011,E2 -17150.011} C_VEL
LIN {X 0,Y 284.35,Z 284.69,A -85,B 0,C 180,E1 -17153.616,E2 -17153.616} C_VEL
LIN {X 0,Y 284.302,Z 284.696,A -85,B 0,C 180,E1 -17157.188,E2 -17157.188} C_VEL
LIN {X 0,Y 284.355,Z 284.686,A -85,B 0,C 180,E1 -17160.375,E2 -17160.375} C_VEL
LIN {X 0,Y 284.374,Z 284.689,A -85,B 0,C 180,E1 -17163.585,E2 -17163.585} C_VEL
LIN {X 0,Y 284.359,Z 284.689,A -85,B 0,C 180,E1 -17166.705,E2 -17166.705} C_VEL
LIN {X 0,Y 284.396,Z 284.687,A -85,B 0,C 180,E1 -17171.26,E2 -17171.26} C_VEL
LIN {X 0,Y 284.484,Z 284.672,A -85,B 0,C 180,E1 -17174.458,E2 -17174.458} C_VEL
LIN {X 0,Y 284.481,Z 284.671,A -85,B 0,C 180,E1 -17178.6,E2 -17178.6} C_VEL
LIN {X 0,Y 284.649,Z 284.646,A -85,B 0,C 180,E1 -17181.48,E2 -17181.48} C_VEL
LIN {X 0,Y 284.548,Z 284.665,A -85,B 0,C 180,E1 -17184.329,E2 -17184.329} C_VEL
LIN {X 0,Y 284.195,Z 284.754,A -85,B 0,C 180,E1 -17186.898,E2 -17186.898} C_VEL
LIN {X 0,Y 285.191,Z 287.592,A -85,B 0,C 180,E1 -17187.136,E2 -17187.136} C_VEL
LIN {X 0,Y 286.627,Z 290.034,A -85,B 0,C 180,E1 -17187.417,E2 -17187.417} C_VEL
LIN {X 0,Y 289.066,Z 294.837,A -85,B 0,C 180,E1 -17187.935,E2 -17187.935} C_VEL
LIN {X 0,Y 294.291,Z 308.936,A -85,B 0,C 180,E1 -17189.358,E2 -17189.358} C_VEL
LIN {X 0,Y 298.054,Z 319.201,A -85,B 0,C 180,E1 -17190.543,E2 -17190.543} C_VEL
LIN {X 0,Y 301.434,Z 331.182,A -85,B 0,C 180,E1 -17191.964,E2 -17191.964} C_VEL
LIN {X 0,Y 302.882,Z 338.33,A -85,B 0,C 180,E1 -17192.842,E2 -17192.842} C_VEL
LIN {X 0,Y 300.655,Z 351.69,A -85,B 0,C 180,E1 -17194.188,E2 -17194.188} C_VEL
LIN {X 0,Y 298.11,Z 365.08,A -85,B 0,C 180,E1 -17195.86,E2 -17195.86} C_VEL
LIN {X 0,Y 295.653,Z 377.004,A -85,B 0,C 180,E1 -17197.683,E2 -17197.683} C_VEL
LIN {X 0,Y 293.195,Z 387.772,A -85,B 0,C 180,E1 -17199.659,E2 -17199.659} C_VEL
LIN {X 0,Y 290.852,Z 397.702,A -85,B 0,C 180,E1 -17201.851,E2 -17201.851} C_VEL
LIN {X 0,Y 288.481,Z 407.369,A -85,B 0,C 180,E1 -17204.459,E2 -17204.459} C_VEL
LIN {X 0,Y 286.66,Z 415.323,A -85,B 0,C 180,E1 -17207.109,E2 -17207.109} C_VEL
LIN {X 0,Y 285.295,Z 421.013,A -85,B 0,C 180,E1 -17209.423,E2 -17209.423} C_VEL
LIN {X 0,Y 284.273,Z 425.713,A -85,B 0,C 180,E1 -17211.766,E2 -17211.766} C_VEL
LIN {X 0,Y 283.686,Z 428.68,A -85,B 0,C 180,E1 -17213.567,E2 -17213.567} C_VEL
LIN {X 0,Y 282.957,Z 432.522,A -85,B 0,C 180,E1 -17216.604,E2 -17216.604} C_VEL
LIN {X 0,Y 282.483,Z 435.115,A -85,B 0,C 180,E1 -17219.839,E2 -17219.839} C_VEL
LIN {X 0,Y 282.391,Z 436.094,A -85,B 0,C 180,E1 -17222.206,E2 -17222.206} C_VEL
LIN {X 0,Y 282.436,Z 436.225,A -85,B 0,C 180,E1 -17224.911,E2 -17224.911} C_VEL
LIN {X 0,Y 282.626,Z 435.509,A -85,B 0,C 180,E1 -17227.279,E2 -17227.279} C_VEL
LIN {X 0,Y 283.22,Z 433.585,A -85,B 0,C 180,E1 -17230.178,E2 -17230.178} C_VEL
LIN {X 0,Y 284.054,Z 430.686,A -85,B 0,C 180,E1 -17232.872,E2 -17232.872} C_VEL
LIN {X 0,Y 285.177,Z 426.561,A -85,B 0,C 180,E1 -17235.616,E2 -17235.616} C_VEL
LIN {X 0,Y 286.899,Z 420.643,A -85,B 0,C 180,E1 -17238.596,E2 -17238.596} C_VEL
LIN {X 0,Y 289.161,Z 413.082,A -85,B 0,C 180,E1 -17241.542,E2 -17241.542} C_VEL
LIN {X 0,Y 291.386,Z 405.524,A -85,B 0,C 180,E1 -17243.898,E2 -17243.898} C_VEL
LIN {X 0,Y 293.933,Z 396.658,A -85,B 0,C 180,E1 -17246.187,E2 -17246.187} C_VEL
LIN {X 0,Y 296.915,Z 386.007,A -85,B 0,C 180,E1 -17248.441,E2 -17248.441} C_VEL
LIN {X 0,Y 299.895,Z 374.755,A -85,B 0,C 180,E1 -17250.394,E2 -17250.394} C_VEL
LIN {X 0,Y 302.486,Z 363.747,A -85,B 0,C 180,E1 -17251.991,E2 -17251.991} C_VEL
LIN {X 0,Y 305.285,Z 350.665,A -85,B 0,C 180,E1 -17253.546,E2 -17253.546} C_VEL
LIN {X 0,Y 306.812,Z 342.322,A -85,B 0,C 180,E1 -17254.384,E2 -17254.384} C_VEL
LIN {X 0,Y 303.567,Z 329.556,A -85,B 0,C 180,E1 -17256.235,E2 -17256.235} C_VEL
LIN {X 0,Y 300.113,Z 319.329,A -85,B 0,C 180,E1 -17257.71,E2 -17257.71} C_VEL
LIN {X 0,Y 294.764,Z 306.997,A -85,B 0,C 180,E1 -17259.532,E2 -17259.532} C_VEL
LIN {X 0,Y 289.487,Z 297.213,A -85,B 0,C 180,E1 -17261.085,E2 -17261.085} C_VEL
LIN {X 0,Y 287.305,Z 293.437,A -85,B 0,C 180,E1 -17261.69,E2 -17261.69} C_VEL
LIN {X 0,Y 285.493,Z 290.88,A -85,B 0,C 180,E1 -17262.173,E2 -17262.173} C_VEL
LIN {X 0,Y 284.884,Z 288.935,A -85,B 0,C 180,E1 -17262.412,E2 -17262.412} C_VEL
LIN {X 0,Y 284.896,Z 287.495,A -85,B 0,C 180,E1 -17265.72,E2 -17265.72} C_VEL
LIN {X 0,Y 284.801,Z 285.624,A -85,B 0,C 180,E1 -17270.771,E2 -17270.771} C_VEL
LIN {X 0,Y 284.7,Z 284.892,A -85,B 0,C 180,E1 -17273.146,E2 -17273.146} C_VEL
LIN {X 0,Y 283.939,Z 284.811,A -85,B 0,C 180,E1 -17274.326,E2 -17274.326} C_VEL
LIN {X 0,Y 281.122,Z 285.091,A -85,B 0,C 180,E1 -17276.254,E2 -17276.254} C_VEL
LIN {X 0,Y 278.827,Z 285.376,A -85,B 0,C 180,E1 -17277.819,E2 -17277.819} C_VEL
LIN {X 0,Y 277.889,Z 285.496,A -85,B 0,C 180,E1 -17279.03,E2 -17279.03} C_VEL
LIN {X 0,Y 277.833,Z 285.497,A -85,B 0,C 180,E1 -17279.439,E2 -17279.439} C_VEL
LIN {X 0,Y 277.696,Z 285.52,A -85,B 0,C 180,E1 -17282.903,E2 -17282.903} C_VEL
LIN {X 0,Y 277.649,Z 285.526,A -85,B 0,C 180,E1 -17287.272,E2 -17287.272} C_VEL
LIN {X 0,Y 277.503,Z 285.54,A -85,B 0,C 180,E1 -17290.213,E2 -17290.213} C_VEL
LIN {X 0,Y 277.432,Z 285.547,A -85,B 0,C 180,E1 -17294.676,E2 -17294.676} C_VEL
LIN {X 0,Y 277.434,Z 285.606,A -85,B 0,C 180,E1 -17296.181,E2 -17296.181} C_VEL
LIN {X 0,Y 277.574,Z 287.046,A -85,B 0,C 180,E1 -17300.762,E2 -17300.762} C_VEL
LIN {X 0,Y 277.854,Z 288.623,A -85,B 0,C 180,E1 -17304.417,E2 -17304.417} C_VEL
LIN {X 0,Y 278.199,Z 290.444,A -85,B 0,C 180,E1 -17307.851,E2 -17307.851} C_VEL
LIN {X 0,Y 278.571,Z 293.147,A -85,B 0,C 180,E1 -17311.994,E2 -17311.994} C_VEL
LIN {X 0,Y 279.182,Z 296.476,A -85,B 0,C 180,E1 -17316.338,E2 -17316.338} C_VEL
LIN {X 0,Y 279.787,Z 300.46,A -85,B 0,C 180,E1 -17320.777,E2 -17320.777} C_VEL
LIN {X 0,Y 280.491,Z 304.274,A -85,B 0,C 180,E1 -17324.555,E2 -17324.555} C_VEL
LIN {X 0,Y 280.703,Z 307.543,A -85,B 0,C 180,E1 -17327.47,E2 -17327.47} C_VEL
LIN {X 0,Y 280.279,Z 310.155,A -85,B 0,C 180,E1 -17329.572,E2 -17329.572} C_VEL
LIN {X 0,Y 281.281,Z 313.517,A -85,B 0,C 180,E1 -17329.923,E2 -17329.923} C_VEL
LIN {X 0,Y 282.544,Z 316.042,A -85,B 0,C 180,E1 -17330.3,E2 -17330.3} C_VEL
LIN {X 0,Y 286.328,Z 325.888,A -85,B 0,C 180,E1 -17331.554,E2 -17331.554} C_VEL
LIN {X 0,Y 290.297,Z 338.228,A -85,B 0,C 180,E1 -17333.078,E2 -17333.078} C_VEL
LIN {X 0,Y 293.214,Z 350.633,A -85,B 0,C 180,E1 -17334.583,E2 -17334.583} C_VEL
LIN {X 0,Y 295.181,Z 363.873,A -85,B 0,C 180,E1 -17336.195,E2 -17336.195} C_VEL
LIN {X 0,Y 295.967,Z 376.449,A -85,B 0,C 180,E1 -17337.789,E2 -17337.789} C_VEL
LIN {X 0,Y 295.895,Z 385.885,A -85,B 0,C 180,E1 -17339.06,E2 -17339.06} C_VEL
LIN {X 0,Y 292.711,Z 398.843,A -85,B 0,C 180,E1 -17340.713,E2 -17340.713} C_VEL
LIN {X 0,Y 289.515,Z 410.588,A -85,B 0,C 180,E1 -17342.535,E2 -17342.535} C_VEL
LIN {X 0,Y 286.499,Z 421.435,A -85,B 0,C 180,E1 -17344.579,E2 -17344.579} C_VEL
LIN {X 0,Y 283.607,Z 432.076,A -85,B 0,C 180,E1 -17347.028,E2 -17347.028} C_VEL
LIN {X 0,Y 281.03,Z 441.008,A -85,B 0,C 180,E1 -17349.507,E2 -17349.507} C_VEL
LIN {X 0,Y 279.316,Z 447.512,A -85,B 0,C 180,E1 -17351.669,E2 -17351.669} C_VEL
LIN {X 0,Y 277.425,Z 454.989,A -85,B 0,C 180,E1 -17354.697,E2 -17354.697} C_VEL
LIN {X 0,Y 276.36,Z 460.453,A -85,B 0,C 180,E1 -17357.517,E2 -17357.517} C_VEL
LIN {X 0,Y 275.796,Z 463.909,A -85,B 0,C 180,E1 -17359.726,E2 -17359.726} C_VEL
LIN {X 0,Y 275.488,Z 467.358,A -85,B 0,C 180,E1 -17362.673,E2 -17362.673} C_VEL
LIN {X 0,Y 275.492,Z 468.692,A -85,B 0,C 180,E1 -17364.229,E2 -17364.229} C_VEL
LIN {X 0,Y 275.412,Z 470.251,A -85,B 0,C 180,E1 -17367.076,E2 -17367.076} C_VEL
LIN {X 0,Y 275.472,Z 470.714,A -85,B 0,C 180,E1 -17370.001,E2 -17370.001} C_VEL
LIN {X 0,Y 275.413,Z 469.993,A -85,B 0,C 180,E1 -17372.926,E2 -17372.926} C_VEL
LIN {X 0,Y 275.493,Z 468.063,A -85,B 0,C 180,E1 -17375.858,E2 -17375.858} C_VEL
LIN {X 0,Y 275.635,Z 464.852,A -85,B 0,C 180,E1 -17378.801,E2 -17378.801} C_VEL
LIN {X 0,Y 276.112,Z 460.344,A -85,B 0,C 180,E1 -17381.75,E2 -17381.75} C_VEL
LIN {X 0,Y 277.157,Z 454.44,A -85,B 0,C 180,E1 -17384.69,E2 -17384.69} C_VEL
LIN {X 0,Y 278.741,Z 446.981,A -85,B 0,C 180,E1 -17387.612,E2 -17387.612} C_VEL
LIN {X 0,Y 280.566,Z 438.991,A -85,B 0,C 180,E1 -17390.148,E2 -17390.148} C_VEL
LIN {X 0,Y 282.978,Z 429.411,A -85,B 0,C 180,E1 -17392.642,E2 -17392.642} C_VEL
LIN {X 0,Y 285.308,Z 419.632,A -85,B 0,C 180,E1 -17394.757,E2 -17394.757} C_VEL
LIN {X 0,Y 288.123,Z 408.05,A -85,B 0,C 180,E1 -17396.825,E2 -17396.825} C_VEL
LIN {X 0,Y 290.992,Z 395.315,A -85,B 0,C 180,E1 -17398.688,E2 -17398.688} C_VEL
LIN {X 0,Y 293.606,Z 382.814,A -85,B 0,C 180,E1 -17400.178,E2 -17400.178} C_VEL
LIN {X 0,Y 292.417,Z 369.545,A -85,B 0,C 180,E1 -17401.822,E2 -17401.822} C_VEL
LIN {X 0,Y 290.368,Z 355.374,A -85,B 0,C 180,E1 -17403.381,E2 -17403.381} C_VEL
LIN {X 0,Y 287.001,Z 339.384,A -85,B 0,C 180,E1 -17404.956,E2 -17404.956} C_VEL
LIN {X 0,Y 282.479,Z 323.692,A -85,B 0,C 180,E1 -17406.351,E2 -17406.351} C_VEL
LIN {X 0,Y 279.423,Z 314.113,A -85,B 0,C 180,E1 -17407.11,E2 -17407.11} C_VEL
LIN {X 0,Y 279.351,Z 313.549,A -85,B 0,C 180,E1 -17407.144,E2 -17407.144} C_VEL
LIN {X 0,Y 280.233,Z 308.679,A -85,B 0,C 180,E1 -17410.698,E2 -17410.698} C_VEL
LIN {X 0,Y 280.55,Z 305.13,A -85,B 0,C 180,E1 -17413.407,E2 -17413.407} C_VEL
LIN {X 0,Y 280.28,Z 302.649,A -85,B 0,C 180,E1 -17415.403,E2 -17415.403} C_VEL
LIN {X 0,Y 279.421,Z 298.304,A -85,B 0,C 180,E1 -17419.158,E2 -17419.158} C_VEL
LIN {X 0,Y 278.711,Z 294.377,A -85,B 0,C 180,E1 -17422.756,E2 -17422.756} C_VEL
LIN {X 0,Y 278.117,Z 290.523,A -85,B 0,C 180,E1 -17426.504,E2 -17426.504} C_VEL
LIN {X 0,Y 277.634,Z 287.595,A -85,B 0,C 180,E1 -17429.582,E2 -17429.582} C_VEL
LIN {X 0,Y 277.299,Z 285.571,A -85,B 0,C 180,E1 -17431.926,E2 -17431.926} C_VEL
LIN {X 0,Y 277.335,Z 285.566,A -85,B 0,C 180,E1 -17436.079,E2 -17436.079} C_VEL
LIN {X 0,Y 277.352,Z 285.562,A -85,B 0,C 180,E1 -17440.765,E2 -17440.765} C_VEL
LIN {X 0,Y 277.441,Z 285.551,A -85,B 0,C 180,E1 -17445.325,E2 -17445.325} C_VEL
LIN {X 0,Y 277.466,Z 285.548,A -85,B 0,C 180,E1 -17449.786,E2 -17449.786} C_VEL
LIN {X 0,Y 277.616,Z 285.531,A -85,B 0,C 180,E1 -17452.727,E2 -17452.727} C_VEL
LIN {X 0,Y 277.826,Z 285.505,A -85,B 0,C 180,E1 -17458.549,E2 -17458.549} C_VEL
LIN {X 0,Y 277.826,Z 285.5,A -85,B 0,C 180,E1 -17461.448,E2 -17461.448} C_VEL
LIN {X 0,Y 277.657,Z 285.521,A -85,B 0,C 180,E1 -17467.269,E2 -17467.269} C_VEL
LIN {X 0,Y 277.51,Z 285.539,A -85,B 0,C 180,E1 -17470.209,E2 -17470.209} C_VEL
LIN {X 0,Y 277.437,Z 285.549,A -85,B 0,C 180,E1 -17474.672,E2 -17474.672} C_VEL
LIN {X 0,Y 277.346,Z 285.554,A -85,B 0,C 180,E1 -17479.232,E2 -17479.232} C_VEL
LIN {X 0,Y 277.32,Z 285.568,A -85,B 0,C 180,E1 -17484.168,E2 -17484.168} C_VEL
LIN {X 0,Y 277.323,Z 285.559,A -85,B 0,C 180,E1 -17487.502,E2 -17487.502} C_VEL
LIN {X 0,Y 277.271,Z 285.57,A -85,B 0,C 180,E1 -17490.479,E2 -17490.479} C_VEL
LIN {X 0,Y 277.253,Z 285.572,A -85,B 0,C 180,E1 -17493.893,E2 -17493.893} C_VEL
LIN {X 0,Y 277.278,Z 285.566,A -85,B 0,C 180,E1 -17497.465,E2 -17497.465} C_VEL
LIN {X 0,Y 277.23,Z 285.574,A -85,B 0,C 180,E1 -17501.23,E2 -17501.23} C_VEL
LIN {X 0,Y 277.243,Z 285.573,A -85,B 0,C 180,E1 -17505.215,E2 -17505.215} C_VEL
LIN {X 0,Y 277.29,Z 285.563,A -85,B 0,C 180,E1 -17509.492,E2 -17509.492} C_VEL
LIN {X 0,Y 277.285,Z 285.568,A -85,B 0,C 180,E1 -17512.532,E2 -17512.532} C_VEL
LIN {X 0,Y 277.248,Z 285.575,A -85,B 0,C 180,E1 -17516.103,E2 -17516.103} C_VEL
LIN {X 0,Y 277.255,Z 285.573,A -85,B 0,C 180,E1 -17519.537,E2 -17519.537} C_VEL
LIN {X 0,Y 277.356,Z 285.562,A -85,B 0,C 180,E1 -17522.863,E2 -17522.863} C_VEL
LIN {X 0,Y 277.321,Z 285.567,A -85,B 0,C 180,E1 -17526.078,E2 -17526.078} C_VEL
LIN {X 0,Y 277.337,Z 285.563,A -85,B 0,C 180,E1 -17530.765,E2 -17530.765} C_VEL
LIN {X 0,Y 277.426,Z 285.552,A -85,B 0,C 180,E1 -17535.324,E2 -17535.324} C_VEL
LIN {X 0,Y 277.498,Z 285.545,A -85,B 0,C 180,E1 -17539.787,E2 -17539.787} C_VEL
LIN {X 0,Y 277.641,Z 285.514,A -85,B 0,C 180,E1 -17542.728,E2 -17542.728} C_VEL
LIN {X 0,Y 277.205,Z 285.581,A -85,B 0,C 180,E1 -17545.956,E2 -17545.956} C_VEL
LIN {X 0,Y 278.131,Z 288.32,A -85,B 0,C 180,E1 -17546.211,E2 -17546.211} C_VEL
LIN {X 0,Y 279.596,Z 290.862,A -85,B 0,C 180,E1 -17546.514,E2 -17546.514} C_VEL
LIN {X 0,Y 283.617,Z 298.547,A -85,B 0,C 180,E1 -17547.416,E2 -17547.416} C_VEL
LIN {X 0,Y 288.59,Z 312.524,A -85,B 0,C 180,E1 -17548.915,E2 -17548.915} C_VEL
LIN {X 0,Y 292.224,Z 322.681,A -85,B 0,C 180,E1 -17550.14,E2 -17550.14} C_VEL
LIN {X 0,Y 295.632,Z 335.665,A -85,B 0,C 180,E1 -17551.772,E2 -17551.772} C_VEL
LIN {X 0,Y 296.334,Z 340.172,A -85,B 0,C 180,E1 -17552.344,E2 -17552.344} C_VEL
LIN {X 0,Y 294.092,Z 353.348,A -85,B 0,C 180,E1 -17553.733,E2 -17553.733} C_VEL
LIN {X 0,Y 291.554,Z 365.993,A -85,B 0,C 180,E1 -17555.359,E2 -17555.359} C_VEL
LIN {X 0,Y 289.102,Z 377.475,A -85,B 0,C 180,E1 -17557.156,E2 -17557.156} C_VEL
LIN {X 0,Y 286.558,Z 388.236,A -85,B 0,C 180,E1 -17559.172,E2 -17559.172} C_VEL
LIN {X 0,Y 284.132,Z 398.158,A -85,B 0,C 180,E1 -17561.412,E2 -17561.412} C_VEL
LIN {X 0,Y 281.734,Z 407.47,A -85,B 0,C 180,E1 -17563.965,E2 -17563.965} C_VEL
LIN {X 0,Y 279.868,Z 415.257,A -85,B 0,C 180,E1 -17566.587,E2 -17566.587} C_VEL
LIN {X 0,Y 278.322,Z 421.473,A -85,B 0,C 180,E1 -17569.162,E2 -17569.162} C_VEL
LIN {X 0,Y 277.281,Z 426.163,A -85,B 0,C 180,E1 -17571.561,E2 -17571.561} C_VEL
LIN {X 0,Y 276.475,Z 430.009,A -85,B 0,C 180,E1 -17573.998,E2 -17573.998} C_VEL
LIN {X 0,Y 275.794,Z 433.354,A -85,B 0,C 180,E1 -17576.892,E2 -17576.892} C_VEL
LIN {X 0,Y 275.398,Z 435.551,A -85,B 0,C 180,E1 -17579.817,E2 -17579.817} C_VEL
LIN {X 0,Y 275.297,Z 436.591,A -85,B 0,C 180,E1 -17582.604,E2 -17582.604} C_VEL
LIN {X 0,Y 275.359,Z 436.661,A -85,B 0,C 180,E1 -17585.244,E2 -17585.244} C_VEL
LIN {X 0,Y 275.627,Z 435.801,A -85,B 0,C 180,E1 -17587.776,E2 -17587.776} C_VEL
LIN {X 0,Y 276.151,Z 434.221,A -85,B 0,C 180,E1 -17590.23,E2 -17590.23} C_VEL
LIN {X 0,Y 277.096,Z 431.112,A -85,B 0,C 180,E1 -17593.219,E2 -17593.219} C_VEL
LIN {X 0,Y 278.301,Z 426.985,A -85,B 0,C 180,E1 -17596.029,E2 -17596.029} C_VEL
LIN {X 0,Y 279.975,Z 421.551,A -85,B 0,C 180,E1 -17598.855,E2 -17598.855} C_VEL
LIN {X 0,Y 281.955,Z 415.237,A -85,B 0,C 180,E1 -17601.456,E2 -17601.456} C_VEL
LIN {X 0,Y 284.326,Z 407.743,A -85,B 0,C 180,E1 -17603.961,E2 -17603.961} C_VEL
LIN {X 0,Y 286.985,Z 398.991,A -85,B 0,C 180,E1 -17606.368,E2 -17606.368} C_VEL
LIN {X 0,Y 290.038,Z 388.777,A -85,B 0,C 180,E1 -17608.664,E2 -17608.664} C_VEL
LIN {X 0,Y 293.148,Z 377.746,A -85,B 0,C 180,E1 -17610.697,E2 -17610.697} C_VEL
LIN {X 0,Y 296.127,Z 365.924,A -85,B 0,C 180,E1 -17612.499,E2 -17612.499} C_VEL
LIN {X 0,Y 298.967,Z 353.512,A -85,B 0,C 180,E1 -17614.043,E2 -17614.043} C_VEL
LIN {X 0,Y 300.679,Z 344.934,A -85,B 0,C 180,E1 -17614.943,E2 -17614.943} C_VEL
LIN {X 0,Y 298.57,Z 335.202,A -85,B 0,C 180,E1 -17616.414,E2 -17616.414} C_VEL
LIN {X 0,Y 295.517,Z 324.952,A -85,B 0,C 180,E1 -17617.957,E2 -17617.957} C_VEL
LIN {X 0,Y 290.31,Z 312.155,A -85,B 0,C 180,E1 -17619.97,E2 -17619.97} C_VEL
LIN {X 0,Y 284.916,Z 301.672,A -85,B 0,C 180,E1 -17621.718,E2 -17621.718} C_VEL
LIN {X 0,Y 282.656,Z 297.885,A -85,B 0,C 180,E1 -17622.409,E2 -17622.409} C_VEL
LIN {X 0,Y 280.28,Z 293.99,A -85,B 0,C 180,E1 -17623.102,E2 -17623.102} C_VEL
LIN {X 0,Y 278.478,Z 291.395,A -85,B 0,C 180,E1 -17623.631,E2 -17623.631} C_VEL
LIN {X 0,Y 277.97,Z 289.588,A -85,B 0,C 180,E1 -17623.893,E2 -17623.893} C_VEL
LIN {X 0,Y 277.812,Z 287.879,A -85,B 0,C 180,E1 -17628.325,E2 -17628.325} C_VEL
LIN {X 0,Y 277.846,Z 286.889,A -85,B 0,C 180,E1 -17631.272,E2 -17631.272} C_VEL
LIN {X 0,Y 277.67,Z 286.076,A -85,B 0,C 180,E1 -17634.191,E2 -17634.191} C_VEL
LIN {X 0,Y 277.696,Z 285.52,A -85,B 0,C 180,E1 -17637.1,E2 -17637.1} C_VEL
LIN {X 0,Y 277.833,Z 285.497,A -85,B 0,C 180,E1 -17639.439,E2 -17639.439} C_VEL
LIN {X 0,Y 277.163,Z 285.585,A -85,B 0,C 180,E1 -17640.647,E2 -17640.647} C_VEL
LIN {X 0,Y 274.125,Z 285.963,A -85,B 0,C 180,E1 -17642.609,E2 -17642.609} C_VEL
LIN {X 0,Y 271.576,Z 286.278,A -85,B 0,C 180,E1 -17644.204,E2 -17644.204} C_VEL
LIN {X 0,Y 270.563,Z 286.408,A -85,B 0,C 180,E1 -17645.446,E2 -17645.446} C_VEL
LIN {X 0,Y 270.526,Z 286.408,A -85,B 0,C 180,E1 -17645.867,E2 -17645.867} C_VEL
LIN {X 0,Y 270.59,Z 286.403,A -85,B 0,C 180,E1 -17649.267,E2 -17649.267} C_VEL
LIN {X 0,Y 270.402,Z 286.731,A -85,B 0,C 180,E1 -17653.529,E2 -17653.529} C_VEL
LIN {X 0,Y 270.537,Z 287.4,A -85,B 0,C 180,E1 -17656.606,E2 -17656.606} C_VEL
LIN {X 0,Y 270.708,Z 288.947,A -85,B 0,C 180,E1 -17661.314,E2 -17661.314} C_VEL
LIN {X 0,Y 270.979,Z 290.474,A -85,B 0,C 180,E1 -17664.807,E2 -17664.807} C_VEL
LIN {X 0,Y 271.319,Z 292.324,A -85,B 0,C 180,E1 -17668.275,E2 -17668.275} C_VEL
LIN {X 0,Y 271.601,Z 294.277,A -85,B 0,C 180,E1 -17671.362,E2 -17671.362} C_VEL
LIN {X 0,Y 271.98,Z 296.639,A -85,B 0,C 180,E1 -17674.646,E2 -17674.646} C_VEL
LIN {X 0,Y 272.445,Z 299.596,A -85,B 0,C 180,E1 -17678.252,E2 -17678.252} C_VEL
LIN {X 0,Y 273.022,Z 303.048,A -85,B 0,C 180,E1 -17682.013,E2 -17682.013} C_VEL
LIN {X 0,Y 273.586,Z 305.988,A -85,B 0,C 180,E1 -17684.946,E2 -17684.946} C_VEL
LIN {X 0,Y 273.69,Z 308.948,A -85,B 0,C 180,E1 -17687.62,E2 -17687.62} C_VEL
LIN {X 0,Y 273.616,Z 309.459,A -85,B 0,C 180,E1 -17688.056,E2 -17688.056} C_VEL
LIN {X 0,Y 274.757,Z 313.061,A -85,B 0,C 180,E1 -17688.504,E2 -17688.504} C_VEL
LIN {X 0,Y 275.969,Z 315.354,A -85,B 0,C 180,E1 -17688.89,E2 -17688.89} C_VEL
LIN {X 0,Y 277.581,Z 319.234,A -85,B 0,C 180,E1 -17689.427,E2 -17689.427} C_VEL
LIN {X 0,Y 281.449,Z 329.729,A -85,B 0,C 180,E1 -17690.863,E2 -17690.863} C_VEL
LIN {X 0,Y 285.009,Z 341.692,A -85,B 0,C 180,E1 -17692.437,E2 -17692.437} C_VEL
LIN {X 0,Y 287.762,Z 354.786,A -85,B 0,C 180,E1 -17694.117,E2 -17694.117} C_VEL
LIN {X 0,Y 289.388,Z 368.378,A -85,B 0,C 180,E1 -17695.87,E2 -17695.87} C_VEL
LIN {X 0,Y 289.808,Z 378.498,A -85,B 0,C 180,E1 -17697.234,E2 -17697.234} C_VEL
LIN {X 0,Y 289.658,Z 386.998,A -85,B 0,C 180,E1 -17698.436,E2 -17698.436} C_VEL
LIN {X 0,Y 286.218,Z 400.126,A -85,B 0,C 180,E1 -17700.184,E2 -17700.184} C_VEL
LIN {X 0,Y 282.637,Z 412.548,A -85,B 0,C 180,E1 -17702.211,E2 -17702.211} C_VEL
LIN {X 0,Y 279.584,Z 423.002,A -85,B 0,C 180,E1 -17704.304,E2 -17704.304} C_VEL
LIN {X 0,Y 276.98,Z 431.94,A -85,B 0,C 180,E1 -17706.446,E2 -17706.446} C_VEL
LIN {X 0,Y 274.325,Z 440.807,A -85,B 0,C 180,E1 -17708.983,E2 -17708.983} C_VEL
LIN {X 0,Y 272.499,Z 447.269,A -85,B 0,C 180,E1 -17711.194,E2 -17711.194} C_VEL
LIN {X 0,Y 270.546,Z 454.4,A -85,B 0,C 180,E1 -17714.162,E2 -17714.162} C_VEL
LIN {X 0,Y 269.375,Z 460.127,A -85,B 0,C 180,E1 -17717.188,E2 -17717.188} C_VEL
LIN {X 0,Y 268.762,Z 463.548,A -85,B 0,C 180,E1 -17719.454,E2 -17719.454} C_VEL
LIN {X 0,Y 268.394,Z 466.984,A -85,B 0,C 180,E1 -17722.478,E2 -17722.478} C_VEL
LIN {X 0,Y 268.416,Z 468.443,A -85,B 0,C 180,E1 -17724.256,E2 -17724.256} C_VEL
LIN {X 0,Y 268.341,Z 469.831,A -85,B 0,C 180,E1 -17726.998,E2 -17726.998} C_VEL
LIN {X 0,Y 268.387,Z 470.267,A -85,B 0,C 180,E1 -17730.001,E2 -17730.001} C_VEL
LIN {X 0,Y 268.343,Z 469.519,A -85,B 0,C 180,E1 -17733.004,E2 -17733.004} C_VEL
LIN {X 0,Y 268.4,Z 467.569,A -85,B 0,C 180,E1 -17736.013,E2 -17736.013} C_VEL
LIN {X 0,Y 268.584,Z 464.331,A -85,B 0,C 180,E1 -17739.034,E2 -17739.034} C_VEL
LIN {X 0,Y 269.1,Z 459.787,A -85,B 0,C 180,E1 -17742.061,E2 -17742.061} C_VEL
LIN {X 0,Y 270.188,Z 453.839,A -85,B 0,C 180,E1 -17745.078,E2 -17745.078} C_VEL
LIN {X 0,Y 271.879,Z 446.333,A -85,B 0,C 180,E1 -17748.072,E2 -17748.072} C_VEL
LIN {X 0,Y 273.839,Z 438.292,A -85,B 0,C 180,E1 -17750.665,E2 -17750.665} C_VEL
LIN {X 0,Y 276.354,Z 428.646,A -85,B 0,C 180,E1 -17753.216,E2 -17753.216} C_VEL
LIN {X 0,Y 278.769,Z 418.797,A -85,B 0,C 180,E1 -17755.379,E2 -17755.379} C_VEL
LIN {X 0,Y 281.735,Z 407.142,A -85,B 0,C 180,E1 -17757.484,E2 -17757.484} C_VEL
LIN {X 0,Y 284.425,Z 395.606,A -85,B 0,C 180,E1 -17759.211,E2 -17759.211} C_VEL
LIN {X 0,Y 286.886,Z 384.758,A -85,B 0,C 180,E1 -17760.551,E2 -17760.551} C_VEL
LIN {X 0,Y 286.181,Z 373.471,A -85,B 0,C 180,E1 -17762.014,E2 -17762.014} C_VEL
LIN {X 0,Y 284.31,Z 358.777,A -85,B 0,C 180,E1 -17763.742,E2 -17763.742} C_VEL
LIN {X 0,Y 281.228,Z 343.008,A -85,B 0,C 180,E1 -17765.391,E2 -17765.391} C_VEL
LIN {X 0,Y 276.909,Z 327.166,A -85,B 0,C 180,E1 -17766.899,E2 -17766.899} C_VEL
LIN {X 0,Y 272.61,Z 313.812,A -85,B 0,C 180,E1 -17768.056,E2 -17768.056} C_VEL
LIN {X 0,Y 272.56,Z 313.037,A -85,B 0,C 180,E1 -17768.174,E2 -17768.174} C_VEL
LIN {X 0,Y 273.225,Z 309.372,A -85,B 0,C 180,E1 -17770.913,E2 -17770.913} C_VEL
LIN {X 0,Y 273.525,Z 306.791,A -85,B 0,C 180,E1 -17772.915,E2 -17772.915} C_VEL
LIN {X 0,Y 273.348,Z 304.243,A -85,B 0,C 180,E1 -17775.003,E2 -17775.003} C_VEL
LIN {X 0,Y 272.606,Z 300.363,A -85,B 0,C 180,E1 -17778.388,E2 -17778.388} C_VEL
LIN {X 0,Y 271.958,Z 296.809,A -85,B 0,C 180,E1 -17781.667,E2 -17781.667} C_VEL
LIN {X 0,Y 271.24,Z 292.379,A -85,B 0,C 180,E1 -17786.012,E2 -17786.012} C_VEL
LIN {X 0,Y 270.558,Z 288.288,A -85,B 0,C 180,E1 -17790.425,E2 -17790.425} C_VEL
LIN {X 0,Y 270.3,Z 286.443,A -85,B 0,C 180,E1 -17792.531,E2 -17792.531} C_VEL
LIN {X 0,Y 270.284,Z 286.444,A -85,B 0,C 180,E1 -17795.518,E2 -17795.518} C_VEL
LIN {X 0,Y 270.308,Z 286.44,A -85,B 0,C 180,E1 -17800.244,E2 -17800.244} C_VEL
LIN {X 0,Y 270.409,Z 286.429,A -85,B 0,C 180,E1 -17804.934,E2 -17804.934} C_VEL
LIN {X 0,Y 270.418,Z 286.426,A -85,B 0,C 180,E1 -17809.517,E2 -17809.517} C_VEL
LIN {X 0,Y 270.576,Z 286.409,A -85,B 0,C 180,E1 -17812.536,E2 -17812.536} C_VEL
LIN {X 0,Y 270.792,Z 286.381,A -85,B 0,C 180,E1 -17818.511,E2 -17818.511} C_VEL
LIN {X 0,Y 270.791,Z 286.377,A -85,B 0,C 180,E1 -17821.486,E2 -17821.486} C_VEL
LIN {X 0,Y 270.615,Z 286.398,A -85,B 0,C 180,E1 -17827.459,E2 -17827.459} C_VEL
LIN {X 0,Y 270.445,Z 286.416,A -85,B 0,C 180,E1 -17830.479,E2 -17830.479} C_VEL
LIN {X 0,Y 270.405,Z 286.424,A -85,B 0,C 180,E1 -17835.063,E2 -17835.063} C_VEL
LIN {X 0,Y 270.303,Z 286.431,A -85,B 0,C 180,E1 -17839.753,E2 -17839.753} C_VEL
LIN {X 0,Y 270.275,Z 286.442,A -85,B 0,C 180,E1 -17844.583,E2 -17844.583} C_VEL
LIN {X 0,Y 270.27,Z 286.435,A -85,B 0,C 180,E1 -17847.907,E2 -17847.907} C_VEL
LIN {X 0,Y 270.183,Z 286.453,A -85,B 0,C 180,E1 -17851.346,E2 -17851.346} C_VEL
LIN {X 0,Y 270.213,Z 286.443,A -85,B 0,C 180,E1 -17854.901,E2 -17854.901} C_VEL
LIN {X 0,Y 270.22,Z 286.448,A -85,B 0,C 180,E1 -17858.715,E2 -17858.715} C_VEL
LIN {X 0,Y 270.192,Z 286.442,A -85,B 0,C 180,E1 -17862.552,E2 -17862.552} C_VEL
LIN {X 0,Y 270.209,Z 286.449,A -85,B 0,C 180,E1 -17866.738,E2 -17866.738} C_VEL
LIN {X 0,Y 270.242,Z 286.44,A -85,B 0,C 180,E1 -17869.445,E2 -17869.445} C_VEL
LIN {X 0,Y 270.252,Z 286.444,A -85,B 0,C 180,E1 -17873.719,E2 -17873.719} C_VEL
LIN {X 0,Y 270.198,Z 286.452,A -85,B 0,C 180,E1 -17876.891,E2 -17876.891} C_VEL
LIN {X 0,Y 270.23,Z 286.445,A -85,B 0,C 180,E1 -17880.386,E2 -17880.386} C_VEL
LIN {X 0,Y 270.259,Z 286.445,A -85,B 0,C 180,E1 -17883.762,E2 -17883.762} C_VEL
LIN {X 0,Y 270.225,Z 286.451,A -85,B 0,C 180,E1 -17887.037,E2 -17887.037} C_VEL
LIN {X 0,Y 270.294,Z 286.441,A -85,B 0,C 180,E1 -17890.243,E2 -17890.243} C_VEL
LIN {X 0,Y 270.395,Z 286.429,A -85,B 0,C 180,E1 -17894.934,E2 -17894.934} C_VEL
LIN {X 0,Y 270.433,Z 286.425,A -85,B 0,C 180,E1 -17899.518,E2 -17899.518} C_VEL
LIN {X 0,Y 270.599,Z 286.39,A -85,B 0,C 180,E1 -17902.537,E2 -17902.537} C_VEL
LIN {X 0,Y 270.27,Z 286.445,A -85,B 0,C 180,E1 -17905.011,E2 -17905.011} C_VEL
LIN {X 0,Y 271.243,Z 289.324,A -85,B 0,C 180,E1 -17905.282,E2 -17905.282} C_VEL
LIN {X 0,Y 272.666,Z 291.807,A -85,B 0,C 180,E1 -17905.59,E2 -17905.59} C_VEL
LIN {X 0,Y 278.117,Z 302.201,A -85,B 0,C 180,E1 -17906.878,E2 -17906.878} C_VEL
LIN {X 0,Y 282.513,Z 315.025,A -85,B 0,C 180,E1 -17908.328,E2 -17908.328} C_VEL
LIN {X 0,Y 286.179,Z 325.581,A -85,B 0,C 180,E1 -17909.683,E2 -17909.683} C_VEL
LIN {X 0,Y 289.461,Z 338.603,A -85,B 0,C 180,E1 -17911.39,E2 -17911.39} C_VEL
LIN {X 0,Y 289.919,Z 340.835,A -85,B 0,C 180,E1 -17911.7,E2 -17911.7} C_VEL
LIN {X 0,Y 287.704,Z 354.124,A -85,B 0,C 180,E1 -17913.15,E2 -17913.15} C_VEL
LIN {X 0,Y 284.829,Z 367.727,A -85,B 0,C 180,E1 -17914.953,E2 -17914.953} C_VEL
LIN {X 0,Y 282.161,Z 379.713,A -85,B 0,C 180,E1 -17916.921,E2 -17916.921} C_VEL
LIN {X 0,Y 279.522,Z 390.429,A -85,B 0,C 180,E1 -17919.04,E2 -17919.04} C_VEL
LIN {X 0,Y 277.021,Z 400.083,A -85,B 0,C 180,E1 -17921.338,E2 -17921.338} C_VEL
LIN {X 0,Y 274.83,Z 408.238,A -85,B 0,C 180,E1 -17923.662,E2 -17923.662} C_VEL
LIN {X 0,Y 272.835,Z 416.245,A -85,B 0,C 180,E1 -17926.459,E2 -17926.459} C_VEL
LIN {X 0,Y 271.369,Z 421.931,A -85,B 0,C 180,E1 -17928.887,E2 -17928.887} C_VEL
LIN {X 0,Y 270.269,Z 426.62,A -85,B 0,C 180,E1 -17931.348,E2 -17931.348} C_VEL
LIN {X 0,Y 269.218,Z 431.499,A -85,B 0,C 180,E1 -17934.687,E2 -17934.687} C_VEL
LIN {X 0,Y 268.637,Z 434.173,A -85,B 0,C 180,E1 -17937.195,E2 -17937.195} C_VEL
LIN {X 0,Y 268.303,Z 436.214,A -85,B 0,C 180,E1 -17940.189,E2 -17940.189} C_VEL
LIN {X 0,Y 268.211,Z 437.146,A -85,B 0,C 180,E1 -17943.384,E2 -17943.384} C_VEL
LIN {X 0,Y 268.311,Z 437.038,A -85,B 0,C 180,E1 -17945.712,E2 -17945.712} C_VEL
LIN {X 0,Y 268.74,Z 435.809,A -85,B 0,C 180,E1 -17948.875,E2 -17948.875} C_VEL
LIN {X 0,Y 269.215,Z 434.406,A -85,B 0,C 180,E1 -17950.798,E2 -17950.798} C_VEL
LIN {X 0,Y 270.017,Z 431.962,A -85,B 0,C 180,E1 -17953.219,E2 -17953.219} C_VEL
LIN {X 0,Y 271.46,Z 427.422,A -85,B 0,C 180,E1 -17956.46,E2 -17956.46} C_VEL
LIN {X 0,Y 273.142,Z 422.227,A -85,B 0,C 180,E1 -17959.237,E2 -17959.237} C_VEL
LIN {X 0,Y 275.552,Z 415.014,A -85,B 0,C 180,E1 -17962.259,E2 -17962.259} C_VEL
LIN {X 0,Y 277.97,Z 407.731,A -85,B 0,C 180,E1 -17964.712,E2 -17964.712} C_VEL
LIN {X 0,Y 280.795,Z 398.945,A -85,B 0,C 180,E1 -17967.15,E2 -17967.15} C_VEL
LIN {X 0,Y 283.986,Z 388.729,A -85,B 0,C 180,E1 -17969.465,E2 -17969.465} C_VEL
LIN {X 0,Y 286.924,Z 378.795,A -85,B 0,C 180,E1 -17971.333,E2 -17971.333} C_VEL
LIN {X 0,Y 290.067,Z 366.931,A -85,B 0,C 180,E1 -17973.191,E2 -17973.191} C_VEL
LIN {X 0,Y 293.29,Z 353.489,A -85,B 0,C 180,E1 -17974.893,E2 -17974.893} C_VEL
LIN {X 0,Y 294.606,Z 346.226,A -85,B 0,C 180,E1 -17975.702,E2 -17975.702} C_VEL
LIN {X 0,Y 291.703,Z 333.686,A -85,B 0,C 180,E1 -17977.701,E2 -17977.701} C_VEL
LIN {X 0,Y 287.644,Z 321.845,A -85,B 0,C 180,E1 -17979.626,E2 -17979.626} C_VEL
LIN {X 0,Y 282.926,Z 311.062,A -85,B 0,C 180,E1 -17981.467,E2 -17981.467} C_VEL
LIN {X 0,Y 278.559,Z 303.09,A -85,B 0,C 180,E1 -17982.947,E2 -17982.947} C_VEL
LIN {X 0,Y 276.342,Z 299.266,A -85,B 0,C 180,E1 -17983.69,E2 -17983.69} C_VEL
LIN {X 0,Y 274.292,Z 295.948,A -85,B 0,C 180,E1 -17984.349,E2 -17984.349} C_VEL
LIN {X 0,Y 273.303,Z 294.686,A -85,B 0,C 180,E1 -17984.648,E2 -17984.648} C_VEL
LIN {X 0,Y 271.574,Z 292.195,A -85,B 0,C 180,E1 -17985.195,E2 -17985.195} C_VEL
LIN {X 0,Y 270.951,Z 290.315,A -85,B 0,C 180,E1 -17985.449,E2 -17985.449} C_VEL
LIN {X 0,Y 270.882,Z 288.607,A -85,B 0,C 180,E1 -17990.362,E2 -17990.362} C_VEL
LIN {X 0,Y 270.736,Z 287.598,A -85,B 0,C 180,E1 -17994.042,E2 -17994.042} C_VEL
LIN {X 0,Y 270.817,Z 286.631,A -85,B 0,C 180,E1 -17998.515,E2 -17998.515} C_VEL
LIN {X 0,Y 270.783,Z 286.378,A -85,B 0,C 180,E1 -18001.489,E2 -18001.489} C_VEL
LIN {X 0,Y 270.526,Z 286.408,A -85,B 0,C 180,E1 -18005.867,E2 -18005.867} C_VEL
LIN {X 0,Y 269.98,Z 286.538,A -85,B 0,C 180,E1 -18007.11,E2 -18007.11} C_VEL
LIN {X 0,Y 268.442,Z 286.874,A -85,B 0,C 180,E1 -18008.328,E2 -18008.328} C_VEL
LIN {X 0,Y 264.675,Z 287.772,A -85,B 0,C 180,E1 -18010.775,E2 -18010.775} C_VEL
LIN {X 0,Y 263.584,Z 288.143,A -85,B 0,C 180,E1 -18012.051,E2 -18012.051} C_VEL
LIN {X 0,Y 263.486,Z 288.231,A -85,B 0,C 180,E1 -18012.484,E2 -18012.484} C_VEL
LIN {X 0,Y 263.651,Z 289.013,A -85,B 0,C 180,E1 -18016.34,E2 -18016.34} C_VEL
LIN {X 0,Y 263.824,Z 290.577,A -85,B 0,C 180,E1 -18021.197,E2 -18021.197} C_VEL
LIN {X 0,Y 264.103,Z 292.329,A -85,B 0,C 180,E1 -18025.211,E2 -18025.211} C_VEL
LIN {X 0,Y 264.426,Z 294.204,A -85,B 0,C 180,E1 -18028.71,E2 -18028.71} C_VEL
LIN {X 0,Y 264.708,Z 296.342,A -85,B 0,C 180,E1 -18032.075,E2 -18032.075} C_VEL
LIN {X 0,Y 265.18,Z 298.953,A -85,B 0,C 180,E1 -18035.668,E2 -18035.668} C_VEL
LIN {X 0,Y 265.749,Z 302.507,A -85,B 0,C 180,E1 -18039.923,E2 -18039.923} C_VEL
LIN {X 0,Y 266.559,Z 306.961,A -85,B 0,C 180,E1 -18044.614,E2 -18044.614} C_VEL
LIN {X 0,Y 266.727,Z 308.805,A -85,B 0,C 180,E1 -18046.373,E2 -18046.373} C_VEL
LIN {X 0,Y 267.75,Z 311.962,A -85,B 0,C 180,E1 -18046.783,E2 -18046.783} C_VEL
LIN {X 0,Y 269.566,Z 314.974,A -85,B 0,C 180,E1 -18047.389,E2 -18047.389} C_VEL
LIN {X 0,Y 273.692,Z 325.299,A -85,B 0,C 180,E1 -18048.966,E2 -18048.966} C_VEL
LIN {X 0,Y 277.476,Z 336.519,A -85,B 0,C 180,E1 -18050.583,E2 -18050.583} C_VEL
LIN {X 0,Y 280.716,Z 349.806,A -85,B 0,C 180,E1 -18052.413,E2 -18052.413} C_VEL
LIN {X 0,Y 282.56,Z 361.028,A -85,B 0,C 180,E1 -18053.936,E2 -18053.936} C_VEL
LIN {X 0,Y 283.575,Z 373.745,A -85,B 0,C 180,E1 -18055.686,E2 -18055.686} C_VEL
LIN {X 0,Y 283.498,Z 386.982,A -85,B 0,C 180,E1 -18057.611,E2 -18057.611} C_VEL
LIN {X 0,Y 282.754,Z 390.693,A -85,B 0,C 180,E1 -18058.117,E2 -18058.117} C_VEL
LIN {X 0,Y 279.055,Z 403.569,A -85,B 0,C 180,E1 -18059.965,E2 -18059.965} C_VEL
LIN {X 0,Y 275.769,Z 414.432,A -85,B 0,C 180,E1 -18061.871,E2 -18061.871} C_VEL
LIN {X 0,Y 272.671,Z 424.55,A -85,B 0,C 180,E1 -18064.014,E2 -18064.014} C_VEL
LIN {X 0,Y 269.661,Z 434.53,A -85,B 0,C 180,E1 -18066.582,E2 -18066.582} C_VEL
LIN {X 0,Y 266.633,Z 443.967,A -85,B 0,C 180,E1 -18069.56,E2 -18069.56} C_VEL
LIN {X 0,Y 264.615,Z 450.802,A -85,B 0,C 180,E1 -18072.217,E2 -18072.217} C_VEL
LIN {X 0,Y 262.927,Z 457.153,A -85,B 0,C 180,E1 -18075.291,E2 -18075.291} C_VEL
LIN {X 0,Y 261.878,Z 462.125,A -85,B 0,C 180,E1 -18078.389,E2 -18078.389} C_VEL
LIN {X 0,Y 261.457,Z 465.056,A -85,B 0,C 180,E1 -18080.72,E2 -18080.72} C_VEL
LIN {X 0,Y 261.306,Z 467.842,A -85,B 0,C 180,E1 -18083.825,E2 -18083.825} C_VEL
LIN {X 0,Y 261.271,Z 469.414,A -85,B 0,C 180,E1 -18086.917,E2 -18086.917} C_VEL
LIN {X 0,Y 261.305,Z 469.817,A -85,B 0,C 180,E1 -18090.001,E2 -18090.001} C_VEL
LIN {X 0,Y 261.275,Z 469.038,A -85,B 0,C 180,E1 -18093.085,E2 -18093.085} C_VEL
LIN {X 0,Y 261.311,Z 467.058,A -85,B 0,C 180,E1 -18096.177,E2 -18096.177} C_VEL
LIN {X 0,Y 261.509,Z 463.794,A -85,B 0,C 180,E1 -18099.28,E2 -18099.28} C_VEL
LIN {X 0,Y 262.105,Z 459.214,A -85,B 0,C 180,E1 -18102.388,E2 -18102.388} C_VEL
LIN {X 0,Y 263.238,Z 453.221,A -85,B 0,C 180,E1 -18105.486,E2 -18105.486} C_VEL
LIN {X 0,Y 265.037,Z 445.672,A -85,B 0,C 180,E1 -18108.555,E2 -18108.555} C_VEL
LIN {X 0,Y 267.118,Z 437.582,A -85,B 0,C 180,E1 -18111.21,E2 -18111.21} C_VEL
LIN {X 0,Y 269.718,Z 427.978,A -85,B 0,C 180,E1 -18113.795,E2 -18113.795} C_VEL
LIN {X 0,Y 272.283,Z 417.965,A -85,B 0,C 180,E1 -18116.028,E2 -18116.028} C_VEL
LIN {X 0,Y 275.401,Z 406.238,A -85,B 0,C 180,E1 -18118.172,E2 -18118.172} C_VEL
LIN {X 0,Y 278.161,Z 394.6,A -85,B 0,C 180,E1 -18119.935,E2 -18119.935} C_VEL
LIN {X 0,Y 280.292,Z 385.524,A -85,B 0,C 180,E1 -18121.081,E2 -18121.081} C_VEL
LIN {X 0,Y 279.49,Z 373.075,A -85,B 0,C 180,E1 -18122.764,E2 -18122.764} C_VEL
LIN {X 0,Y 277.879,Z 360.061,A -85,B 0,C 180,E1 -18124.35,E2 -18124.35} C_VEL
LIN {X 0,Y 274.987,Z 344.694,A -85,B 0,C 180,E1 -18126.041,E2 -18126.041} C_VEL
LIN {X 0,Y 270.871,Z 329.122,A -85,B 0,C 180,E1 -18127.615,E2 -18127.615} C_VEL
LIN {X 0,Y 266.544,Z 315.887,A -85,B 0,C 180,E1 -18128.842,E2 -18128.842} C_VEL
LIN {X 0,Y 265.713,Z 312.668,A -85,B 0,C 180,E1 -18129.1,E2 -18129.1} C_VEL
LIN {X 0,Y 266.395,Z 308.482,A -85,B 0,C 180,E1 -18132.378,E2 -18132.378} C_VEL
LIN {X 0,Y 266.395,Z 305.832,A -85,B 0,C 180,E1 -18134.575,E2 -18134.575} C_VEL
LIN {X 0,Y 265.56,Z 301.343,A -85,B 0,C 180,E1 -18138.575,E2 -18138.575} C_VEL
LIN {X 0,Y 264.733,Z 296.917,A -85,B 0,C 180,E1 -18142.791,E2 -18142.791} C_VEL
LIN {X 0,Y 264.291,Z 293.704,A -85,B 0,C 180,E1 -18146.051,E2 -18146.051} C_VEL
LIN {X 0,Y 263.714,Z 290.475,A -85,B 0,C 180,E1 -18149.577,E2 -18149.577} C_VEL
LIN {X 0,Y 263.237,Z 287.323,A -85,B 0,C 180,E1 -18153.434,E2 -18153.434} C_VEL
LIN {X 0,Y 263.191,Z 287.329,A -85,B 0,C 180,E1 -18156.386,E2 -18156.386} C_VEL
LIN {X 0,Y 263.27,Z 287.316,A -85,B 0,C 180,E1 -18159.692,E2 -18159.692} C_VEL
LIN {X 0,Y 263.357,Z 287.308,A -85,B 0,C 180,E1 -18164.521,E2 -18164.521} C_VEL
LIN {X 0,Y 263.361,Z 287.306,A -85,B 0,C 180,E1 -18169.232,E2 -18169.232} C_VEL
LIN {X 0,Y 263.538,Z 287.286,A -85,B 0,C 180,E1 -18172.336,E2 -18172.336} C_VEL
LIN {X 0,Y 263.756,Z 287.257,A -85,B 0,C 180,E1 -18178.472,E2 -18178.472} C_VEL
LIN {X 0,Y 263.756,Z 287.253,A -85,B 0,C 180,E1 -18181.525,E2 -18181.525} C_VEL
LIN {X 0,Y 263.577,Z 287.275,A -85,B 0,C 180,E1 -18187.66,E2 -18187.66} C_VEL
LIN {X 0,Y 263.377,Z 287.294,A -85,B 0,C 180,E1 -18190.764,E2 -18190.764} C_VEL
LIN {X 0,Y 263.353,Z 287.303,A -85,B 0,C 180,E1 -18195.476,E2 -18195.476} C_VEL
LIN {X 0,Y 263.265,Z 287.305,A -85,B 0,C 180,E1 -18200.304,E2 -18200.304} C_VEL
LIN {X 0,Y 263.209,Z 287.321,A -85,B 0,C 180,E1 -18205.289,E2 -18205.289} C_VEL
LIN {X 0,Y 263.165,Z 287.32,A -85,B 0,C 180,E1 -18208.729,E2 -18208.729} C_VEL
LIN {X 0,Y 263.132,Z 287.333,A -85,B 0,C 180,E1 -18212.286,E2 -18212.286} C_VEL
LIN {X 0,Y 263.185,Z 287.317,A -85,B 0,C 180,E1 -18215.976,E2 -18215.976} C_VEL
LIN {X 0,Y 263.13,Z 287.335,A -85,B 0,C 180,E1 -18219.865,E2 -18219.865} C_VEL
LIN {X 0,Y 263.136,Z 287.326,A -85,B 0,C 180,E1 -18223.978,E2 -18223.978} C_VEL
LIN {X 0,Y 263.17,Z 287.321,A -85,B 0,C 180,E1 -18228.392,E2 -18228.392} C_VEL
LIN {X 0,Y 263.184,Z 287.327,A -85,B 0,C 180,E1 -18232.106,E2 -18232.106} C_VEL
LIN {X 0,Y 263.178,Z 287.324,A -85,B 0,C 180,E1 -18235.888,E2 -18235.888} C_VEL
LIN {X 0,Y 263.147,Z 287.329,A -85,B 0,C 180,E1 -18239.505,E2 -18239.505} C_VEL
LIN {X 0,Y 263.19,Z 287.328,A -85,B 0,C 180,E1 -18243.001,E2 -18243.001} C_VEL
LIN {X 0,Y 263.177,Z 287.329,A -85,B 0,C 180,E1 -18246.385,E2 -18246.385} C_VEL
LIN {X 0,Y 263.256,Z 287.317,A -85,B 0,C 180,E1 -18249.692,E2 -18249.692} C_VEL
LIN {X 0,Y 263.343,Z 287.306,A -85,B 0,C 180,E1 -18254.52,E2 -18254.52} C_VEL
LIN {X 0,Y 263.366,Z 287.303,A -85,B 0,C 180,E1 -18259.233,E2 -18259.233} C_VEL
LIN {X 0,Y 263.561,Z 287.266,A -85,B 0,C 180,E1 -18262.337,E2 -18262.337} C_VEL
LIN {X 0,Y 263.457,Z 287.291,A -85,B 0,C 180,E1 -18264.018,E2 -18264.018} C_VEL
LIN {X 0,Y 264.468,Z 290.273,A -85,B 0,C 180,E1 -18264.309,E2 -18264.309} C_VEL
LIN {X 0,Y 272.274,Z 305.014,A -85,B 0,C 180,E1 -18266.25,E2 -18266.25} C_VEL
LIN {X 0,Y 276.63,Z 318.054,A -85,B 0,C 180,E1 -18267.8,E2 -18267.8} C_VEL
LIN {X 0,Y 280.316,Z 329.164,A -85,B 0,C 180,E1 -18269.294,E2 -18269.294} C_VEL
LIN {X 0,Y 283.353,Z 341.939,A -85,B 0,C 180,E1 -18271.069,E2 -18271.069} C_VEL
LIN {X 0,Y 283.48,Z 343.296,A -85,B 0,C 180,E1 -18271.244,E2 -18271.244} C_VEL
LIN {X 0,Y 280.764,Z 357.563,A -85,B 0,C 180,E1 -18272.869,E2 -18272.869} C_VEL
LIN {X 0,Y 277.877,Z 370.619,A -85,B 0,C 180,E1 -18274.714,E2 -18274.714} C_VEL
LIN {X 0,Y 275.141,Z 382.215,A -85,B 0,C 180,E1 -18276.728,E2 -18276.728} C_VEL
LIN {X 0,Y 272.076,Z 394.001,A -85,B 0,C 180,E1 -18279.219,E2 -18279.219} C_VEL
LIN {X 0,Y 269.539,Z 403.439,A -85,B 0,C 180,E1 -18281.657,E2 -18281.657} C_VEL
LIN {X 0,Y 267.093,Z 412.348,A -85,B 0,C 180,E1 -18284.474,E2 -18284.474} C_VEL
LIN {X 0,Y 265.134,Z 419.804,A -85,B 0,C 180,E1 -18287.403,E2 -18287.403} C_VEL
LIN {X 0,Y 263.656,Z 425.617,A -85,B 0,C 180,E1 -18290.274,E2 -18290.274} C_VEL
LIN {X 0,Y 262.647,Z 429.703,A -85,B 0,C 180,E1 -18292.829,E2 -18292.829} C_VEL
LIN {X 0,Y 261.938,Z 432.973,A -85,B 0,C 180,E1 -18295.421,E2 -18295.421} C_VEL
LIN {X 0,Y 261.3,Z 435.972,A -85,B 0,C 180,E1 -18298.954,E2 -18298.954} C_VEL
LIN {X 0,Y 261.18,Z 436.904,A -85,B 0,C 180,E1 -18300.747,E2 -18300.747} C_VEL
LIN {X 0,Y 261.137,Z 437.59,A -85,B 0,C 180,E1 -18303.46,E2 -18303.46} C_VEL
LIN {X 0,Y 261.281,Z 437.38,A -85,B 0,C 180,E1 -18306.281,E2 -18306.281} C_VEL
LIN {X 0,Y 261.646,Z 436.409,A -85,B 0,C 180,E1 -18308.838,E2 -18308.838} C_VEL
LIN {X 0,Y 262.497,Z 434.047,A -85,B 0,C 180,E1 -18312.015,E2 -18312.015} C_VEL
LIN {X 0,Y 263.611,Z 430.726,A -85,B 0,C 180,E1 -18314.949,E2 -18314.949} C_VEL
LIN {X 0,Y 265.207,Z 426.204,A -85,B 0,C 180,E1 -18317.901,E2 -18317.901} C_VEL
LIN {X 0,Y 267.248,Z 420.313,A -85,B 0,C 180,E1 -18320.868,E2 -18320.868} C_VEL
LIN {X 0,Y 269.914,Z 412.832,A -85,B 0,C 180,E1 -18323.819,E2 -18323.819} C_VEL
LIN {X 0,Y 272.533,Z 405.216,A -85,B 0,C 180,E1 -18326.267,E2 -18326.267} C_VEL
LIN {X 0,Y 275.639,Z 396.101,A -85,B 0,C 180,E1 -18328.664,E2 -18328.664} C_VEL
LIN {X 0,Y 279.133,Z 385.119,A -85,B 0,C 180,E1 -18331.035,E2 -18331.035} C_VEL
LIN {X 0,Y 282.675,Z 373.204,A -85,B 0,C 180,E1 -18333.115,E2 -18333.115} C_VEL
LIN {X 0,Y 286.028,Z 360.249,A -85,B 0,C 180,E1 -18334.963,E2 -18334.963} C_VEL
LIN {X 0,Y 288.604,Z 349.07,A -85,B 0,C 180,E1 -18336.263,E2 -18336.263} C_VEL
LIN {X 0,Y 286.736,Z 339.509,A -85,B 0,C 180,E1 -18337.863,E2 -18337.863} C_VEL
LIN {X 0,Y 284.18,Z 330.629,A -85,B 0,C 180,E1 -18339.367,E2 -18339.367} C_VEL
LIN {X 0,Y 279.746,Z 318.914,A -85,B 0,C 180,E1 -18341.442,E2 -18341.442} C_VEL
LIN {X 0,Y 274.823,Z 308.766,A -85,B 0,C 180,E1 -18343.367,E2 -18343.367} C_VEL
LIN {X 0,Y 271.27,Z 302.903,A -85,B 0,C 180,E1 -18344.628,E2 -18344.628} C_VEL
LIN {X 0,Y 269.755,Z 300.344,A -85,B 0,C 180,E1 -18345.171,E2 -18345.171} C_VEL
LIN {X 0,Y 267.671,Z 297.092,A -85,B 0,C 180,E1 -18345.908,E2 -18345.908} C_VEL
LIN {X 0,Y 267.048,Z 296.038,A -85,B 0,C 180,E1 -18346.13,E2 -18346.13} C_VEL
LIN {X 0,Y 264.838,Z 293.477,A -85,B 0,C 180,E1 -18346.868,E2 -18346.868} C_VEL
LIN {X 0,Y 263.914,Z 291.033,A -85,B 0,C 180,E1 -18347.311,E2 -18347.311} C_VEL
LIN {X 0,Y 263.941,Z 289.913,A -85,B 0,C 180,E1 -18350.809,E2 -18350.809} C_VEL
LIN {X 0,Y 263.796,Z 289.121,A -85,B 0,C 180,E1 -18353.884,E2 -18353.884} C_VEL
LIN {X 0,Y 263.884,Z 288.201,A -85,B 0,C 180,E1 -18358.476,E2 -18358.476} C_VEL
LIN {X 0,Y 263.828,Z 287.82,A -85,B 0,C 180,E1 -18361.528,E2 -18361.528} C_VEL
LIN {X 0,Y 263.612,Z 287.703,A -85,B 0,C 180,E1 -18367.662,E2 -18367.662} C_VEL
LIN {X 0,Y 263.497,Z 287.971,A -85,B 0,C 180,E1 -18370.762,E2 -18370.762} C_VEL
LIN {X 0,Y 263.486,Z 288.231,A -85,B 0,C 180,E1 -18372.484,E2 -18372.484} C_VEL
LIN {X 0,Y 262.825,Z 288.625,A -85,B 0,C 180,E1 -18373.759,E2 -18373.759} C_VEL
LIN {X 0,Y 260.102,Z 289.753,A -85,B 0,C 180,E1 -18375.835,E2 -18375.835} C_VEL
LIN {X 0,Y 257.816,Z 290.766,A -85,B 0,C 180,E1 -18377.52,E2 -18377.52} C_VEL
LIN {X 0,Y 256.853,Z 291.405,A -85,B 0,C 180,E1 -18378.826,E2 -18378.826} C_VEL
LIN {X 0,Y 256.783,Z 291.57,A -85,B 0,C 180,E1 -18379.268,E2 -18379.268} C_VEL
LIN {X 0,Y 256.969,Z 292.77,A -85,B 0,C 180,E1 -18382.515,E2 -18382.515} C_VEL
LIN {X 0,Y 257.225,Z 294.32,A -85,B 0,C 180,E1 -18385.924,E2 -18385.924} C_VEL
LIN {X 0,Y 257.552,Z 296.229,A -85,B 0,C 180,E1 -18389.42,E2 -18389.42} C_VEL
LIN {X 0,Y 257.876,Z 298.563,A -85,B 0,C 180,E1 -18393.031,E2 -18393.031} C_VEL
LIN {X 0,Y 258.353,Z 301.311,A -85,B 0,C 180,E1 -18396.762,E2 -18396.762} C_VEL
LIN {X 0,Y 258.886,Z 304.582,A -85,B 0,C 180,E1 -18400.659,E2 -18400.659} C_VEL
LIN {X 0,Y 259.531,Z 308.071,A -85,B 0,C 180,E1 -18404.368,E2 -18404.368} C_VEL
LIN {X 0,Y 260.822,Z 311.489,A -85,B 0,C 180,E1 -18404.92,E2 -18404.92} C_VEL
LIN {X 0,Y 262.886,Z 314.369,A -85,B 0,C 180,E1 -18405.657,E2 -18405.657} C_VEL
LIN {X 0,Y 264.746,Z 318.434,A -85,B 0,C 180,E1 -18406.386,E2 -18406.386} C_VEL
LIN {X 0,Y 266.039,Z 321.407,A -85,B 0,C 180,E1 -18406.912,E2 -18406.912} C_VEL
LIN {X 0,Y 269.028,Z 329.187,A -85,B 0,C 180,E1 -18408.19,E2 -18408.19} C_VEL
LIN {X 0,Y 272.712,Z 341.318,A -85,B 0,C 180,E1 -18410.041,E2 -18410.041} C_VEL
LIN {X 0,Y 275.614,Z 354.786,A -85,B 0,C 180,E1 -18412.009,E2 -18412.009} C_VEL
LIN {X 0,Y 277.186,Z 367.701,A -85,B 0,C 180,E1 -18413.861,E2 -18413.861} C_VEL
LIN {X 0,Y 277.571,Z 381.045,A -85,B 0,C 180,E1 -18415.824,E2 -18415.824} C_VEL
LIN {X 0,Y 277.04,Z 389.951,A -85,B 0,C 180,E1 -18417.204,E2 -18417.204} C_VEL
LIN {X 0,Y 273.277,Z 402.655,A -85,B 0,C 180,E1 -18419.047,E2 -18419.047} C_VEL
LIN {X 0,Y 269.501,Z 414.48,A -85,B 0,C 180,E1 -18421.156,E2 -18421.156} C_VEL
LIN {X 0,Y 266.253,Z 424.515,A -85,B 0,C 180,E1 -18423.339,E2 -18423.339} C_VEL
LIN {X 0,Y 263.081,Z 434.404,A -85,B 0,C 180,E1 -18425.96,E2 -18425.96} C_VEL
LIN {X 0,Y 259.922,Z 443.755,A -85,B 0,C 180,E1 -18429.008,E2 -18429.008} C_VEL
LIN {X 0,Y 257.792,Z 450.564,A -85,B 0,C 180,E1 -18431.73,E2 -18431.73} C_VEL
LIN {X 0,Y 255.99,Z 456.873,A -85,B 0,C 180,E1 -18434.883,E2 -18434.883} C_VEL
LIN {X 0,Y 254.866,Z 461.803,A -85,B 0,C 180,E1 -18438.065,E2 -18438.065} C_VEL
LIN {X 0,Y 254.387,Z 464.688,A -85,B 0,C 180,E1 -18440.46,E2 -18440.46} C_VEL
LIN {X 0,Y 254.229,Z 467.456,A -85,B 0,C 180,E1 -18443.653,E2 -18443.653} C_VEL
LIN {X 0,Y 254.202,Z 468.997,A -85,B 0,C 180,E1 -18446.831,E2 -18446.831} C_VEL
LIN {X 0,Y 254.225,Z 469.369,A -85,B 0,C 180,E1 -18450.001,E2 -18450.001} C_VEL
LIN {X 0,Y 254.208,Z 468.557,A -85,B 0,C 180,E1 -18453.171,E2 -18453.171} C_VEL
LIN {X 0,Y 254.233,Z 466.542,A -85,B 0,C 180,E1 -18456.35,E2 -18456.35} C_VEL
LIN {X 0,Y 254.458,Z 463.259,A -85,B 0,C 180,E1 -18459.54,E2 -18459.54} C_VEL
LIN {X 0,Y 255.117,Z 458.64,A -85,B 0,C 180,E1 -18462.733,E2 -18462.733} C_VEL
LIN {X 0,Y 256.305,Z 452.604,A -85,B 0,C 180,E1 -18465.916,E2 -18465.916} C_VEL
LIN {X 0,Y 258.209,Z 445.01,A -85,B 0,C 180,E1 -18469.065,E2 -18469.065} C_VEL
LIN {X 0,Y 260.45,Z 436.875,A -85,B 0,C 180,E1 -18471.78,E2 -18471.78} C_VEL
LIN {X 0,Y 263.012,Z 427.628,A -85,B 0,C 180,E1 -18474.322,E2 -18474.322} C_VEL
LIN {X 0,Y 265.837,Z 417.116,A -85,B 0,C 180,E1 -18476.708,E2 -18476.708} C_VEL
LIN {X 0,Y 269.07,Z 405.295,A -85,B 0,C 180,E1 -18478.897,E2 -18478.897} C_VEL
LIN {X 0,Y 271.65,Z 394.837,A -85,B 0,C 180,E1 -18480.514,E2 -18480.514} C_VEL
LIN {X 0,Y 273.708,Z 386.247,A -85,B 0,C 180,E1 -18481.634,E2 -18481.634} C_VEL
LIN {X 0,Y 272.916,Z 373.319,A -85,B 0,C 180,E1 -18483.449,E2 -18483.449} C_VEL
LIN {X 0,Y 271.262,Z 360.155,A -85,B 0,C 180,E1 -18485.126,E2 -18485.126} C_VEL
LIN {X 0,Y 268.59,Z 345.616,A -85,B 0,C 180,E1 -18486.804,E2 -18486.804} C_VEL
LIN {X 0,Y 264.57,Z 330.024,A -85,B 0,C 180,E1 -18488.445,E2 -18488.445} C_VEL
LIN {X 0,Y 259.556,Z 314.87,A -85,B 0,C 180,E1 -18489.933,E2 -18489.933} C_VEL
LIN {X 0,Y 258.96,Z 312.198,A -85,B 0,C 180,E1 -18490.162,E2 -18490.162} C_VEL
LIN {X 0,Y 259.418,Z 308.727,A -85,B 0,C 180,E1 -18492.989,E2 -18492.989} C_VEL
LIN {X 0,Y 259.257,Z 306.2,A -85,B 0,C 180,E1 -18495.184,E2 -18495.184} C_VEL
LIN {X 0,Y 258.424,Z 301.779,A -85,B 0,C 180,E1 -18499.253,E2 -18499.253} C_VEL
LIN {X 0,Y 257.683,Z 297.857,A -85,B 0,C 180,E1 -18503.127,E2 -18503.127} C_VEL
LIN {X 0,Y 257.145,Z 294.292,A -85,B 0,C 180,E1 -18506.863,E2 -18506.863} C_VEL
LIN {X 0,Y 256.535,Z 290.438,A -85,B 0,C 180,E1 -18511.245,E2 -18511.245} C_VEL
LIN {X 0,Y 256.193,Z 288.201,A -85,B 0,C 180,E1 -18514.232,E2 -18514.232} C_VEL
LIN {X 0,Y 256.174,Z 288.2,A -85,B 0,C 180,E1 -18519.104,E2 -18519.104} C_VEL
LIN {X 0,Y 256.307,Z 288.185,A -85,B 0,C 180,E1 -18524.084,E2 -18524.084} C_VEL
LIN {X 0,Y 256.301,Z 288.186,A -85,B 0,C 180,E1 -18527.327,E2 -18527.327} C_VEL
LIN {X 0,Y 256.501,Z 288.162,A -85,B 0,C 180,E1 -18532.124,E2 -18532.124} C_VEL
LIN {X 0,Y 256.5,Z 288.16,A -85,B 0,C 180,E1 -18536.857,E2 -18536.857} C_VEL
LIN {X 0,Y 256.771,Z 288.125,A -85,B 0,C 180,E1 -18539.998,E2 -18539.998} C_VEL
LIN {X 0,Y 256.502,Z 288.15,A -85,B 0,C 180,E1 -18543.14,E2 -18543.14} C_VEL
LIN {X 0,Y 256.544,Z 288.152,A -85,B 0,C 180,E1 -18547.871,E2 -18547.871} C_VEL
LIN {X 0,Y 256.313,Z 288.173,A -85,B 0,C 180,E1 -18551.064,E2 -18551.064} C_VEL
LIN {X 0,Y 256.303,Z 288.183,A -85,B 0,C 180,E1 -18555.913,E2 -18555.913} C_VEL
LIN {X 0,Y 256.168,Z 288.191,A -85,B 0,C 180,E1 -18560.893,E2 -18560.893} C_VEL
LIN {X 0,Y 256.189,Z 288.196,A -85,B 0,C 180,E1 -18565.136,E2 -18565.136} C_VEL
LIN {X 0,Y 256.103,Z 288.2,A -85,B 0,C 180,E1 -18569.599,E2 -18569.599} C_VEL
LIN {X 0,Y 256.084,Z 288.209,A -85,B 0,C 180,E1 -18573.288,E2 -18573.288} C_VEL
LIN {X 0,Y 256.127,Z 288.199,A -85,B 0,C 180,E1 -18577.273,E2 -18577.273} C_VEL
LIN {X 0,Y 256.078,Z 288.208,A -85,B 0,C 180,E1 -18581.196,E2 -18581.196} C_VEL
LIN {X 0,Y 256.072,Z 288.211,A -85,B 0,C 180,E1 -18585.524,E2 -18585.524} C_VEL
LIN {X 0,Y 256.1,Z 288.201,A -85,B 0,C 180,E1 -18588.804,E2 -18588.804} C_VEL
LIN {X 0,Y 256.151,Z 288.201,A -85,B 0,C 180,E1 -18592.87,E2 -18592.87} C_VEL
LIN {X 0,Y 256.08,Z 288.21,A -85,B 0,C 180,E1 -18596.708,E2 -18596.708} C_VEL
LIN {X 0,Y 256.136,Z 288.203,A -85,B 0,C 180,E1 -18601.401,E2 -18601.401} C_VEL
LIN {X 0,Y 256.16,Z 288.201,A -85,B 0,C 180,E1 -18605.697,E2 -18605.697} C_VEL
LIN {X 0,Y 256.159,Z 288.199,A -85,B 0,C 180,E1 -18609.103,E2 -18609.103} C_VEL
LIN {X 0,Y 256.292,Z 288.185,A -85,B 0,C 180,E1 -18614.083,E2 -18614.083} C_VEL
LIN {X 0,Y 256.301,Z 288.181,A -85,B 0,C 180,E1 -18618.933,E2 -18618.933} C_VEL
LIN {X 0,Y 256.529,Z 288.141,A -85,B 0,C 180,E1 -18622.126,E2 -18622.126} C_VEL
LIN {X 0,Y 256.498,Z 288.34,A -85,B 0,C 180,E1 -18622.966,E2 -18622.966} C_VEL
LIN {X 0,Y 257.536,Z 291.12,A -85,B 0,C 180,E1 -18623.26,E2 -18623.26} C_VEL
LIN {X 0,Y 258.848,Z 293.322,A -85,B 0,C 180,E1 -18623.568,E2 -18623.568} C_VEL
LIN {X 0,Y 266.304,Z 307.809,A -85,B 0,C 180,E1 -18625.572,E2 -18625.572} C_VEL
LIN {X 0,Y 269.425,Z 316.949,A -85,B 0,C 180,E1 -18626.717,E2 -18626.717} C_VEL
LIN {X 0,Y 274.148,Z 331.502,A -85,B 0,C 180,E1 -18628.732,E2 -18628.732} C_VEL
LIN {X 0,Y 276.916,Z 343.435,A -85,B 0,C 180,E1 -18630.471,E2 -18630.471} C_VEL
LIN {X 0,Y 277.072,Z 344.877,A -85,B 0,C 180,E1 -18630.667,E2 -18630.667} C_VEL
LIN {X 0,Y 274.304,Z 358.775,A -85,B 0,C 180,E1 -18632.308,E2 -18632.308} C_VEL
LIN {X 0,Y 271.462,Z 371.029,A -85,B 0,C 180,E1 -18634.082,E2 -18634.082} C_VEL
LIN {X 0,Y 268.362,Z 383.7,A -85,B 0,C 180,E1 -18636.351,E2 -18636.351} C_VEL
LIN {X 0,Y 265.366,Z 394.716,A -85,B 0,C 180,E1 -18638.758,E2 -18638.758} C_VEL
LIN {X 0,Y 262.817,Z 403.855,A -85,B 0,C 180,E1 -18641.178,E2 -18641.178} C_VEL
LIN {X 0,Y 260.255,Z 412.778,A -85,B 0,C 180,E1 -18644.065,E2 -18644.065} C_VEL
LIN {X 0,Y 258.526,Z 419.106,A -85,B 0,C 180,E1 -18646.584,E2 -18646.584} C_VEL
LIN {X 0,Y 257.012,Z 424.476,A -85,B 0,C 180,E1 -18649.155,E2 -18649.155} C_VEL
LIN {X 0,Y 255.947,Z 428.976,A -85,B 0,C 180,E1 -18651.806,E2 -18651.806} C_VEL
LIN {X 0,Y 255.063,Z 432.61,A -85,B 0,C 180,E1 -18654.6,E2 -18654.6} C_VEL
LIN {X 0,Y 254.331,Z 435.779,A -85,B 0,C 180,E1 -18658.018,E2 -18658.018} C_VEL
LIN {X 0,Y 254.09,Z 437.416,A -85,B 0,C 180,E1 -18660.974,E2 -18660.974} C_VEL
LIN {X 0,Y 254.064,Z 438.09,A -85,B 0,C 180,E1 -18663.919,E2 -18663.919} C_VEL
LIN {X 0,Y 254.339,Z 437.586,A -85,B 0,C 180,E1 -18667.437,E2 -18667.437} C_VEL
LIN {X 0,Y 254.707,Z 436.688,A -85,B 0,C 180,E1 -18669.417,E2 -18669.417} C_VEL
LIN {X 0,Y 255.411,Z 434.792,A -85,B 0,C 180,E1 -18672.021,E2 -18672.021} C_VEL
LIN {X 0,Y 256.732,Z 431.185,A -85,B 0,C 180,E1 -18675.375,E2 -18675.375} C_VEL
LIN {X 0,Y 258.413,Z 426.702,A -85,B 0,C 180,E1 -18678.382,E2 -18678.382} C_VEL
LIN {X 0,Y 260.826,Z 420.177,A -85,B 0,C 180,E1 -18681.706,E2 -18681.706} C_VEL
LIN {X 0,Y 263.627,Z 412.769,A -85,B 0,C 180,E1 -18684.645,E2 -18684.645} C_VEL
LIN {X 0,Y 266.778,Z 403.973,A -85,B 0,C 180,E1 -18687.457,E2 -18687.457} C_VEL
LIN {X 0,Y 270.185,Z 394.339,A -85,B 0,C 180,E1 -18689.941,E2 -18689.941} C_VEL
LIN {X 0,Y 273.765,Z 383.547,A -85,B 0,C 180,E1 -18692.211,E2 -18692.211} C_VEL
LIN {X 0,Y 277.154,Z 372.408,A -85,B 0,C 180,E1 -18694.139,E2 -18694.139} C_VEL
LIN {X 0,Y 280.29,Z 360.951,A -85,B 0,C 180,E1 -18695.79,E2 -18695.79} C_VEL
LIN {X 0,Y 282.628,Z 351.392,A -85,B 0,C 180,E1 -18696.933,E2 -18696.933} C_VEL
LIN {X 0,Y 281.618,Z 345.171,A -85,B 0,C 180,E1 -18698.019,E2 -18698.019} C_VEL
LIN {X 0,Y 279.215,Z 335.481,A -85,B 0,C 180,E1 -18699.753,E2 -18699.753} C_VEL
LIN {X 0,Y 275.153,Z 323.834,A -85,B 0,C 180,E1 -18701.907,E2 -18701.907} C_VEL
LIN {X 0,Y 270.453,Z 313.606,A -85,B 0,C 180,E1 -18703.984,E2 -18703.984} C_VEL
LIN {X 0,Y 265.829,Z 305.535,A -85,B 0,C 180,E1 -18705.806,E2 -18705.806} C_VEL
LIN {X 0,Y 263.156,Z 301.351,A -85,B 0,C 180,E1 -18706.832,E2 -18706.832} C_VEL
LIN {X 0,Y 260.855,Z 298.035,A -85,B 0,C 180,E1 -18707.703,E2 -18707.703} C_VEL
LIN {X 0,Y 260.324,Z 296.978,A -85,B 0,C 180,E1 -18707.925,E2 -18707.925} C_VEL
LIN {X 0,Y 258.001,Z 294.553,A -85,B 0,C 180,E1 -18708.779,E2 -18708.779} C_VEL
LIN {X 0,Y 256.949,Z 291.812,A -85,B 0,C 180,E1 -18709.328,E2 -18709.328} C_VEL
LIN {X 0,Y 256.939,Z 291.04,A -85,B 0,C 180,E1 -18712.141,E2 -18712.141} C_VEL
LIN {X 0,Y 256.836,Z 290.031,A -85,B 0,C 180,E1 -18716.864,E2 -18716.864} C_VEL
LIN {X 0,Y 257.03,Z 289.534,A -85,B 0,C 180,E1 -18720.002,E2 -18720.002} C_VEL
LIN {X 0,Y 256.729,Z 289.347,A -85,B 0,C 180,E1 -18723.14,E2 -18723.14} C_VEL
LIN {X 0,Y 256.696,Z 289.361,A -85,B 0,C 180,E1 -18727.87,E2 -18727.87} C_VEL
LIN {X 0,Y 256.597,Z 289.678,A -85,B 0,C 180,E1 -18731.055,E2 -18731.055} C_VEL
LIN {X 0,Y 256.729,Z 290.58,A -85,B 0,C 180,E1 -18735.889,E2 -18735.889} C_VEL
LIN {X 0,Y 256.783,Z 291.57,A -85,B 0,C 180,E1 -18739.268,E2 -18739.268} C_VEL
LIN {X 0,Y 256.182,Z 292.187,A -85,B 0,C 180,E1 -18740.571,E2 -18740.571} C_VEL
LIN {X 0,Y 253.535,Z 293.689,A -85,B 0,C 180,E1 -18742.69,E2 -18742.69} C_VEL
LIN {X 0,Y 251.301,Z 295,A -85,B 0,C 180,E1 -18744.411,E2 -18744.411} C_VEL
LIN {X 0,Y 250.383,Z 295.861,A -85,B 0,C 180,E1 -18745.744,E2 -18745.744} C_VEL
LIN {X 0,Y 250.33,Z 296.1,A -85,B 0,C 180,E1 -18746.196,E2 -18746.196} C_VEL
LIN {X 0,Y 250.649,Z 297.962,A -85,B 0,C 180,E1 -18749.635,E2 -18749.635} C_VEL
LIN {X 0,Y 251.073,Z 300.809,A -85,B 0,C 180,E1 -18754.046,E2 -18754.046} C_VEL
LIN {X 0,Y 251.554,Z 303.716,A -85,B 0,C 180,E1 -18757.928,E2 -18757.928} C_VEL
LIN {X 0,Y 252.154,Z 307.371,A -85,B 0,C 180,E1 -18762.032,E2 -18762.032} C_VEL
LIN {X 0,Y 253.45,Z 310.618,A -85,B 0,C 180,E1 -18762.654,E2 -18762.654} C_VEL
LIN {X 0,Y 256.076,Z 314.09,A -85,B 0,C 180,E1 -18763.709,E2 -18763.709} C_VEL
LIN {X 0,Y 258.052,Z 318.031,A -85,B 0,C 180,E1 -18764.533,E2 -18764.533} C_VEL
LIN {X 0,Y 259.254,Z 320.035,A -85,B 0,C 180,E1 -18765.022,E2 -18765.022} C_VEL
LIN {X 0,Y 262.123,Z 326.638,A -85,B 0,C 180,E1 -18766.296,E2 -18766.296} C_VEL
LIN {X 0,Y 265.723,Z 337.58,A -85,B 0,C 180,E1 -18768.151,E2 -18768.151} C_VEL
LIN {X 0,Y 268.954,Z 351.032,A -85,B 0,C 180,E1 -18770.268,E2 -18770.268} C_VEL
LIN {X 0,Y 270.793,Z 362.967,A -85,B 0,C 180,E1 -18772.098,E2 -18772.098} C_VEL
LIN {X 0,Y 271.531,Z 375.62,A -85,B 0,C 180,E1 -18774.028,E2 -18774.028} C_VEL
LIN {X 0,Y 271.205,Z 388.208,A -85,B 0,C 180,E1 -18776.023,E2 -18776.023} C_VEL
LIN {X 0,Y 270.896,Z 391.088,A -85,B 0,C 180,E1 -18776.493,E2 -18776.493} C_VEL
LIN {X 0,Y 266.862,Z 403.934,A -85,B 0,C 180,E1 -18778.439,E2 -18778.439} C_VEL
LIN {X 0,Y 263.296,Z 414.549,A -85,B 0,C 180,E1 -18780.41,E2 -18780.41} C_VEL
LIN {X 0,Y 259.346,Z 425.976,A -85,B 0,C 180,E1 -18783.007,E2 -18783.007} C_VEL
LIN {X 0,Y 256.129,Z 435.544,A -85,B 0,C 180,E1 -18785.697,E2 -18785.697} C_VEL
LIN {X 0,Y 252.877,Z 444.614,A -85,B 0,C 180,E1 -18788.821,E2 -18788.821} C_VEL
LIN {X 0,Y 250.426,Z 451.994,A -85,B 0,C 180,E1 -18792.02,E2 -18792.02} C_VEL
LIN {X 0,Y 248.686,Z 457.905,A -85,B 0,C 180,E1 -18795.266,E2 -18795.266} C_VEL
LIN {X 0,Y 247.635,Z 462.498,A -85,B 0,C 180,E1 -18798.542,E2 -18798.542} C_VEL
LIN {X 0,Y 247.159,Z 465.853,A -85,B 0,C 180,E1 -18801.827,E2 -18801.827} C_VEL
LIN {X 0,Y 247.077,Z 467.974,A -85,B 0,C 180,E1 -18805.106,E2 -18805.106} C_VEL
LIN {X 0,Y 247.104,Z 468.895,A -85,B 0,C 180,E1 -18808.371,E2 -18808.371} C_VEL
LIN {X 0,Y 247.147,Z 468.919,A -85,B 0,C 180,E1 -18810.001,E2 -18810.001} C_VEL
LIN {X 0,Y 247.142,Z 468.073,A -85,B 0,C 180,E1 -18813.262,E2 -18813.262} C_VEL
LIN {X 0,Y 247.159,Z 466.019,A -85,B 0,C 180,E1 -18816.532,E2 -18816.532} C_VEL
LIN {X 0,Y 247.395,Z 462.708,A -85,B 0,C 180,E1 -18819.815,E2 -18819.815} C_VEL
LIN {X 0,Y 248.137,Z 458.051,A -85,B 0,C 180,E1 -18823.097,E2 -18823.097} C_VEL
LIN {X 0,Y 249.394,Z 451.963,A -85,B 0,C 180,E1 -18826.369,E2 -18826.369} C_VEL
LIN {X 0,Y 251.414,Z 444.311,A -85,B 0,C 180,E1 -18829.601,E2 -18829.601} C_VEL
LIN {X 0,Y 253.801,Z 436.115,A -85,B 0,C 180,E1 -18832.381,E2 -18832.381} C_VEL
LIN {X 0,Y 256.203,Z 427.637,A -85,B 0,C 180,E1 -18834.769,E2 -18834.769} C_VEL
LIN {X 0,Y 258.906,Z 418.002,A -85,B 0,C 180,E1 -18837.045,E2 -18837.045} C_VEL
LIN {X 0,Y 262.229,Z 406.444,A -85,B 0,C 180,E1 -18839.284,E2 -18839.284} C_VEL
LIN {X 0,Y 264.869,Z 396.26,A -85,B 0,C 180,E1 -18840.938,E2 -18840.938} C_VEL
LIN {X 0,Y 267.13,Z 387.013,A -85,B 0,C 180,E1 -18842.201,E2 -18842.201} C_VEL
LIN {X 0,Y 266.383,Z 374.172,A -85,B 0,C 180,E1 -18844.091,E2 -18844.091} C_VEL
LIN {X 0,Y 264.989,Z 362.128,A -85,B 0,C 180,E1 -18845.697,E2 -18845.697} C_VEL
LIN {X 0,Y 262.749,Z 349.12,A -85,B 0,C 180,E1 -18847.272,E2 -18847.272} C_VEL
LIN {X 0,Y 259.084,Z 333.977,A -85,B 0,C 180,E1 -18848.981,E2 -18848.981} C_VEL
LIN {X 0,Y 254.502,Z 319.122,A -85,B 0,C 180,E1 -18850.543,E2 -18850.543} C_VEL
LIN {X 0,Y 252.202,Z 312.537,A -85,B 0,C 180,E1 -18851.2,E2 -18851.2} C_VEL
LIN {X 0,Y 252.119,Z 311.753,A -85,B 0,C 180,E1 -18851.27,E2 -18851.27} C_VEL
LIN {X 0,Y 252.375,Z 308.438,A -85,B 0,C 180,E1 -18854.123,E2 -18854.123} C_VEL
LIN {X 0,Y 252.009,Z 305.851,A -85,B 0,C 180,E1 -18856.477,E2 -18856.477} C_VEL
LIN {X 0,Y 251.282,Z 302.227,A -85,B 0,C 180,E1 -18859.962,E2 -18859.962} C_VEL
LIN {X 0,Y 250.505,Z 297.842,A -85,B 0,C 180,E1 -18864.451,E2 -18864.451} C_VEL
LIN {X 0,Y 250.032,Z 294.872,A -85,B 0,C 180,E1 -18867.718,E2 -18867.718} C_VEL
LIN {X 0,Y 249.558,Z 291.741,A -85,B 0,C 180,E1 -18871.395,E2 -18871.395} C_VEL
LIN {X 0,Y 249.158,Z 289.077,A -85,B 0,C 180,E1 -18874.968,E2 -18874.968} C_VEL
LIN {X 0,Y 249.118,Z 289.08,A -85,B 0,C 180,E1 -18880.211,E2 -18880.211} C_VEL
LIN {X 0,Y 249.249,Z 289.063,A -85,B 0,C 180,E1 -18883.621,E2 -18883.621} C_VEL
LIN {X 0,Y 249.251,Z 289.067,A -85,B 0,C 180,E1 -18888.615,E2 -18888.615} C_VEL
LIN {X 0,Y 249.444,Z 289.04,A -85,B 0,C 180,E1 -18891.9,E2 -18891.9} C_VEL
LIN {X 0,Y 249.292,Z 289.057,A -85,B 0,C 180,E1 -18895.147,E2 -18895.147} C_VEL
LIN {X 0,Y 249.68,Z 289.01,A -85,B 0,C 180,E1 -18898.385,E2 -18898.385} C_VEL
LIN {X 0,Y 249.68,Z 289.007,A -85,B 0,C 180,E1 -18901.611,E2 -18901.611} C_VEL
LIN {X 0,Y 249.454,Z 289.032,A -85,B 0,C 180,E1 -18906.77,E2 -18906.77} C_VEL
LIN {X 0,Y 249.428,Z 289.038,A -85,B 0,C 180,E1 -18909.731,E2 -18909.731} C_VEL
LIN {X 0,Y 249.208,Z 289.066,A -85,B 0,C 180,E1 -18914.701,E2 -18914.701} C_VEL
LIN {X 0,Y 249.142,Z 289.071,A -85,B 0,C 180,E1 -18918.075,E2 -18918.075} C_VEL
LIN {X 0,Y 249.089,Z 289.072,A -85,B 0,C 180,E1 -18921.516,E2 -18921.516} C_VEL
LIN {X 0,Y 249.131,Z 289.076,A -85,B 0,C 180,E1 -18925.48,E2 -18925.48} C_VEL
LIN {X 0,Y 249.073,Z 289.074,A -85,B 0,C 180,E1 -18928.987,E2 -18928.987} C_VEL
LIN {X 0,Y 249.035,Z 289.088,A -85,B 0,C 180,E1 -18932.423,E2 -18932.423} C_VEL
LIN {X 0,Y 249.067,Z 289.075,A -85,B 0,C 180,E1 -18936.336,E2 -18936.336} C_VEL
LIN {X 0,Y 249.032,Z 289.086,A -85,B 0,C 180,E1 -18940.47,E2 -18940.47} C_VEL
LIN {X 0,Y 249.016,Z 289.088,A -85,B 0,C 180,E1 -18944.873,E2 -18944.873} C_VEL
LIN {X 0,Y 249.059,Z 289.086,A -85,B 0,C 180,E1 -18947.37,E2 -18947.37} C_VEL
LIN {X 0,Y 249.048,Z 289.087,A -85,B 0,C 180,E1 -18951.622,E2 -18951.622} C_VEL
LIN {X 0,Y 249.056,Z 289.08,A -85,B 0,C 180,E1 -18955.64,E2 -18955.64} C_VEL
LIN {X 0,Y 249.047,Z 289.085,A -85,B 0,C 180,E1 -18959.471,E2 -18959.471} C_VEL
LIN {X 0,Y 249.07,Z 289.088,A -85,B 0,C 180,E1 -18963.161,E2 -18963.161} C_VEL
LIN {X 0,Y 249.072,Z 289.086,A -85,B 0,C 180,E1 -18966.731,E2 -18966.731} C_VEL
LIN {X 0,Y 249.103,Z 289.081,A -85,B 0,C 180,E1 -18970.21,E2 -18970.21} C_VEL
LIN {X 0,Y 249.234,Z 289.064,A -85,B 0,C 180,E1 -18973.62,E2 -18973.62} C_VEL
LIN {X 0,Y 249.245,Z 289.06,A -85,B 0,C 180,E1 -18978.615,E2 -18978.615} C_VEL
LIN {X 0,Y 249.479,Z 289.02,A -85,B 0,C 180,E1 -18981.804,E2 -18981.804} C_VEL
LIN {X 0,Y 250.441,Z 291.786,A -85,B 0,C 180,E1 -18982.107,E2 -18982.107} C_VEL
LIN {X 0,Y 252.003,Z 294.264,A -85,B 0,C 180,E1 -18982.49,E2 -18982.49} C_VEL
LIN {X 0,Y 260.034,Z 309.809,A -85,B 0,C 180,E1 -18984.761,E2 -18984.761} C_VEL
LIN {X 0,Y 262.01,Z 314.767,A -85,B 0,C 180,E1 -18985.461,E2 -18985.461} C_VEL
LIN {X 0,Y 265.962,Z 327.528,A -85,B 0,C 180,E1 -18987.218,E2 -18987.218} C_VEL
LIN {X 0,Y 268.853,Z 337.495,A -85,B 0,C 180,E1 -18988.707,E2 -18988.707} C_VEL
LIN {X 0,Y 270.673,Z 345.924,A -85,B 0,C 180,E1 -18989.999,E2 -18989.999} C_VEL
LIN {X 0,Y 267.885,Z 359.822,A -85,B 0,C 180,E1 -18991.701,E2 -18991.701} C_VEL
LIN {X 0,Y 264.81,Z 372.575,A -85,B 0,C 180,E1 -18993.613,E2 -18993.613} C_VEL
LIN {X 0,Y 261.727,Z 384.653,A -85,B 0,C 180,E1 -18995.851,E2 -18995.851} C_VEL
LIN {X 0,Y 258.775,Z 395.124,A -85,B 0,C 180,E1 -18998.196,E2 -18998.196} C_VEL
LIN {X 0,Y 256.025,Z 404.548,A -85,B 0,C 180,E1 -19000.756,E2 -19000.756} C_VEL
LIN {X 0,Y 253.292,Z 413.665,A -85,B 0,C 180,E1 -19003.811,E2 -19003.811} C_VEL
LIN {X 0,Y 251.174,Z 421.106,A -85,B 0,C 180,E1 -19006.929,E2 -19006.929} C_VEL
LIN {X 0,Y 249.665,Z 426.493,A -85,B 0,C 180,E1 -19009.741,E2 -19009.741} C_VEL
LIN {X 0,Y 248.605,Z 430.574,A -85,B 0,C 180,E1 -19012.434,E2 -19012.434} C_VEL
LIN {X 0,Y 247.822,Z 433.853,A -85,B 0,C 180,E1 -19015.174,E2 -19015.174} C_VEL
LIN {X 0,Y 247.138,Z 436.859,A -85,B 0,C 180,E1 -19018.909,E2 -19018.909} C_VEL
LIN {X 0,Y 246.977,Z 437.99,A -85,B 0,C 180,E1 -19021.39,E2 -19021.39} C_VEL
LIN {X 0,Y 246.998,Z 438.521,A -85,B 0,C 180,E1 -19024.684,E2 -19024.684} C_VEL
LIN {X 0,Y 247.239,Z 438.137,A -85,B 0,C 180,E1 -19027.261,E2 -19027.261} C_VEL
LIN {X 0,Y 247.931,Z 436.52,A -85,B 0,C 180,E1 -19030.689,E2 -19030.689} C_VEL
LIN {X 0,Y 248.954,Z 433.98,A -85,B 0,C 180,E1 -19033.758,E2 -19033.758} C_VEL
LIN {X 0,Y 250.417,Z 430.307,A -85,B 0,C 180,E1 -19036.859,E2 -19036.859} C_VEL
LIN {X 0,Y 252.551,Z 424.922,A -85,B 0,C 180,E1 -19040.208,E2 -19040.208} C_VEL
LIN {X 0,Y 254.891,Z 418.966,A -85,B 0,C 180,E1 -19043.09,E2 -19043.09} C_VEL
LIN {X 0,Y 258.058,Z 410.986,A -85,B 0,C 180,E1 -19046.149,E2 -19046.149} C_VEL
LIN {X 0,Y 261.151,Z 402.752,A -85,B 0,C 180,E1 -19048.696,E2 -19048.696} C_VEL
LIN {X 0,Y 264.731,Z 392.989,A -85,B 0,C 180,E1 -19051.17,E2 -19051.17} C_VEL
LIN {X 0,Y 268.564,Z 381.942,A -85,B 0,C 180,E1 -19053.449,E2 -19053.449} C_VEL
LIN {X 0,Y 272.217,Z 370.08,A -85,B 0,C 180,E1 -19055.457,E2 -19055.457} C_VEL
LIN {X 0,Y 275.815,Z 357.082,A -85,B 0,C 180,E1 -19057.235,E2 -19057.235} C_VEL
LIN {X 0,Y 276.721,Z 352.585,A -85,B 0,C 180,E1 -19057.805,E2 -19057.805} C_VEL
LIN {X 0,Y 274.667,Z 342.047,A -85,B 0,C 180,E1 -19059.794,E2 -19059.794} C_VEL
LIN {X 0,Y 271.362,Z 331.195,A -85,B 0,C 180,E1 -19061.895,E2 -19061.895} C_VEL
LIN {X 0,Y 267.371,Z 321.152,A -85,B 0,C 180,E1 -19063.98,E2 -19063.98} C_VEL
LIN {X 0,Y 262.296,Z 311.342,A -85,B 0,C 180,E1 -19066.248,E2 -19066.248} C_VEL
LIN {X 0,Y 259.286,Z 306.609,A -85,B 0,C 180,E1 -19067.516,E2 -19067.516} C_VEL
LIN {X 0,Y 256.597,Z 302.47,A -85,B 0,C 180,E1 -19068.661,E2 -19068.661} C_VEL
LIN {X 0,Y 254.346,Z 299.424,A -85,B 0,C 180,E1 -19069.607,E2 -19069.607} C_VEL
LIN {X 0,Y 253.591,Z 297.895,A -85,B 0,C 180,E1 -19069.955,E2 -19069.955} C_VEL
LIN {X 0,Y 251.199,Z 295.509,A -85,B 0,C 180,E1 -19070.947,E2 -19070.947} C_VEL
LIN {X 0,Y 250,Z 292.651,A -85,B 0,C 180,E1 -19071.616,E2 -19071.616} C_VEL
LIN {X 0,Y 249.81,Z 291.909,A -85,B 0,C 180,E1 -19075.16,E2 -19075.16} C_VEL
LIN {X 0,Y 250.026,Z 291.329,A -85,B 0,C 180,E1 -19078.391,E2 -19078.391} C_VEL
LIN {X 0,Y 250.113,Z 291.118,A -85,B 0,C 180,E1 -19080.002,E2 -19080.002} C_VEL
LIN {X 0,Y 249.822,Z 290.96,A -85,B 0,C 180,E1 -19083.227,E2 -19083.227} C_VEL
LIN {X 0,Y 249.793,Z 291.027,A -85,B 0,C 180,E1 -19088.089,E2 -19088.089} C_VEL
LIN {X 0,Y 249.698,Z 291.388,A -85,B 0,C 180,E1 -19091.364,E2 -19091.364} C_VEL
LIN {X 0,Y 249.769,Z 291.976,A -85,B 0,C 180,E1 -19094.671,E2 -19094.671} C_VEL
LIN {X 0,Y 249.829,Z 292.856,A -85,B 0,C 180,E1 -19098.027,E2 -19098.027} C_VEL
LIN {X 0,Y 250.037,Z 294.208,A -85,B 0,C 180,E1 -19101.946,E2 -19101.946} C_VEL
LIN {X 0,Y 250.33,Z 296.1,A -85,B 0,C 180,E1 -19106.196,E2 -19106.196} C_VEL
LIN {X 0,Y 249.771,Z 296.947,A -85,B 0,C 180,E1 -19107.528,E2 -19107.528} C_VEL
LIN {X 0,Y 247.171,Z 298.799,A -85,B 0,C 180,E1 -19109.691,E2 -19109.691} C_VEL
LIN {X 0,Y 244.973,Z 300.405,A -85,B 0,C 180,E1 -19111.447,E2 -19111.447} C_VEL
LIN {X 0,Y 244.092,Z 301.497,A -85,B 0,C 180,E1 -19112.808,E2 -19112.808} C_VEL
LIN {X 0,Y 244.055,Z 301.816,A -85,B 0,C 180,E1 -19113.27,E2 -19113.27} C_VEL
LIN {X 0,Y 244.491,Z 304.557,A -85,B 0,C 180,E1 -19117.134,E2 -19117.134} C_VEL
LIN {X 0,Y 244.803,Z 306.442,A -85,B 0,C 180,E1 -19119.302,E2 -19119.302} C_VEL
LIN {X 0,Y 245.938,Z 309.416,A -85,B 0,C 180,E1 -19119.948,E2 -19119.948} C_VEL
LIN {X 0,Y 248.343,Z 312.536,A -85,B 0,C 180,E1 -19121.071,E2 -19121.071} C_VEL
LIN {X 0,Y 248.96,Z 313.416,A -85,B 0,C 180,E1 -19121.347,E2 -19121.347} C_VEL
LIN {X 0,Y 250.963,Z 317.331,A -85,B 0,C 180,E1 -19122.299,E2 -19122.299} C_VEL
LIN {X 0,Y 252.542,Z 319.452,A -85,B 0,C 180,E1 -19122.987,E2 -19122.987} C_VEL
LIN {X 0,Y 254.545,Z 323.631,A -85,B 0,C 180,E1 -19123.953,E2 -19123.953} C_VEL
LIN {X 0,Y 255.558,Z 325.59,A -85,B 0,C 180,E1 -19124.405,E2 -19124.405} C_VEL
LIN {X 0,Y 258.286,Z 332.422,A -85,B 0,C 180,E1 -19125.794,E2 -19125.794} C_VEL
LIN {X 0,Y 261.623,Z 344.327,A -85,B 0,C 180,E1 -19127.883,E2 -19127.883} C_VEL
LIN {X 0,Y 263.952,Z 356.067,A -85,B 0,C 180,E1 -19129.821,E2 -19129.821} C_VEL
LIN {X 0,Y 265.221,Z 366.567,A -85,B 0,C 180,E1 -19131.519,E2 -19131.519} C_VEL
LIN {X 0,Y 265.627,Z 377.665,A -85,B 0,C 180,E1 -19133.305,E2 -19133.305} C_VEL
LIN {X 0,Y 265.09,Z 389.411,A -85,B 0,C 180,E1 -19135.274,E2 -19135.274} C_VEL
LIN {X 0,Y 264.504,Z 393.212,A -85,B 0,C 180,E1 -19135.888,E2 -19135.888} C_VEL
LIN {X 0,Y 260.475,Z 405.248,A -85,B 0,C 180,E1 -19137.801,E2 -19137.801} C_VEL
LIN {X 0,Y 256.485,Z 416.462,A -85,B 0,C 180,E1 -19139.997,E2 -19139.997} C_VEL
LIN {X 0,Y 252.466,Z 427.479,A -85,B 0,C 180,E1 -19142.658,E2 -19142.658} C_VEL
LIN {X 0,Y 249.158,Z 436.691,A -85,B 0,C 180,E1 -19145.416,E2 -19145.416} C_VEL
LIN {X 0,Y 245.828,Z 445.476,A -85,B 0,C 180,E1 -19148.624,E2 -19148.624} C_VEL
LIN {X 0,Y 243.617,Z 451.771,A -85,B 0,C 180,E1 -19151.499,E2 -19151.499} C_VEL
LIN {X 0,Y 241.752,Z 457.627,A -85,B 0,C 180,E1 -19154.834,E2 -19154.834} C_VEL
LIN {X 0,Y 240.613,Z 462.163,A -85,B 0,C 180,E1 -19158.203,E2 -19158.203} C_VEL
LIN {X 0,Y 240.077,Z 465.473,A -85,B 0,C 180,E1 -19161.585,E2 -19161.585} C_VEL
LIN {X 0,Y 240.012,Z 467.581,A -85,B 0,C 180,E1 -19164.962,E2 -19164.962} C_VEL
LIN {X 0,Y 240.032,Z 468.465,A -85,B 0,C 180,E1 -19168.323,E2 -19168.323} C_VEL
LIN {X 0,Y 240.071,Z 468.468,A -85,B 0,C 180,E1 -19170.001,E2 -19170.001} C_VEL
LIN {X 0,Y 240.056,Z 467.58,A -85,B 0,C 180,E1 -19173.358,E2 -19173.358} C_VEL
LIN {X 0,Y 240.065,Z 465.483,A -85,B 0,C 180,E1 -19176.726,E2 -19176.726} C_VEL
LIN {X 0,Y 240.35,Z 462.137,A -85,B 0,C 180,E1 -19180.106,E2 -19180.106} C_VEL
LIN {X 0,Y 241.139,Z 457.447,A -85,B 0,C 180,E1 -19183.484,E2 -19183.484} C_VEL
LIN {X 0,Y 242.645,Z 450.81,A -85,B 0,C 180,E1 -19187.092,E2 -19187.092} C_VEL
LIN {X 0,Y 244.642,Z 443.605,A -85,B 0,C 180,E1 -19190.167,E2 -19190.167} C_VEL
LIN {X 0,Y 247.164,Z 435.351,A -85,B 0,C 180,E1 -19193.016,E2 -19193.016} C_VEL
LIN {X 0,Y 249.806,Z 426.007,A -85,B 0,C 180,E1 -19195.681,E2 -19195.681} C_VEL
LIN {X 0,Y 253.081,Z 415.3,A -85,B 0,C 180,E1 -19198.171,E2 -19198.171} C_VEL
LIN {X 0,Y 256.213,Z 404.358,A -85,B 0,C 180,E1 -19200.268,E2 -19200.268} C_VEL
LIN {X 0,Y 259.09,Z 393.907,A -85,B 0,C 180,E1 -19201.936,E2 -19201.936} C_VEL
LIN {X 0,Y 260.571,Z 387.783,A -85,B 0,C 180,E1 -19202.797,E2 -19202.797} C_VEL
LIN {X 0,Y 259.875,Z 375.007,A -85,B 0,C 180,E1 -19204.76,E2 -19204.76} C_VEL
LIN {X 0,Y 258.531,Z 363.014,A -85,B 0,C 180,E1 -19206.415,E2 -19206.415} C_VEL
LIN {X 0,Y 256.479,Z 350.621,A -85,B 0,C 180,E1 -19208.001,E2 -19208.001} C_VEL
LIN {X 0,Y 253.016,Z 335.64,A -85,B 0,C 180,E1 -19209.788,E2 -19209.788} C_VEL
LIN {X 0,Y 248.364,Z 320.268,A -85,B 0,C 180,E1 -19211.487,E2 -19211.487} C_VEL
LIN {X 0,Y 245.315,Z 311.904,A -85,B 0,C 180,E1 -19212.391,E2 -19212.391} C_VEL
LIN {X 0,Y 245.239,Z 311.294,A -85,B 0,C 180,E1 -19212.479,E2 -19212.479} C_VEL
LIN {X 0,Y 245.339,Z 309.273,A -85,B 0,C 180,E1 -19214.261,E2 -19214.261} C_VEL
LIN {X 0,Y 245.007,Z 306.912,A -85,B 0,C 180,E1 -19216.492,E2 -19216.492} C_VEL
LIN {X 0,Y 244.053,Z 302.36,A -85,B 0,C 180,E1 -19221.036,E2 -19221.036} C_VEL
LIN {X 0,Y 243.488,Z 298.864,A -85,B 0,C 180,E1 -19224.739,E2 -19224.739} C_VEL
LIN {X 0,Y 242.911,Z 295.454,A -85,B 0,C 180,E1 -19228.614,E2 -19228.614} C_VEL
LIN {X 0,Y 242.463,Z 292.371,A -85,B 0,C 180,E1 -19232.368,E2 -19232.368} C_VEL
LIN {X 0,Y 242.089,Z 289.957,A -85,B 0,C 180,E1 -19235.562,E2 -19235.562} C_VEL
LIN {X 0,Y 242.045,Z 289.96,A -85,B 0,C 180,E1 -19239.607,E2 -19239.607} C_VEL
LIN {X 0,Y 242.17,Z 289.946,A -85,B 0,C 180,E1 -19243.277,E2 -19243.277} C_VEL
LIN {X 0,Y 242.187,Z 289.946,A -85,B 0,C 180,E1 -19248.278,E2 -19248.278} C_VEL
LIN {X 0,Y 242.394,Z 289.918,A -85,B 0,C 180,E1 -19251.663,E2 -19251.663} C_VEL
LIN {X 0,Y 242.252,Z 289.935,A -85,B 0,C 180,E1 -19255.005,E2 -19255.005} C_VEL
LIN {X 0,Y 242.641,Z 289.887,A -85,B 0,C 180,E1 -19258.338,E2 -19258.338} C_VEL
LIN {X 0,Y 242.641,Z 289.884,A -85,B 0,C 180,E1 -19261.658,E2 -19261.658} C_VEL
LIN {X 0,Y 242.432,Z 289.909,A -85,B 0,C 180,E1 -19266.749,E2 -19266.749} C_VEL
LIN {X 0,Y 242.349,Z 289.918,A -85,B 0,C 180,E1 -19270.018,E2 -19270.018} C_VEL
LIN {X 0,Y 242.17,Z 289.941,A -85,B 0,C 180,E1 -19275.139,E2 -19275.139} C_VEL
LIN {X 0,Y 242.075,Z 289.947,A -85,B 0,C 180,E1 -19278.622,E2 -19278.622} C_VEL
LIN {X 0,Y 242.014,Z 289.957,A -85,B 0,C 180,E1 -19282.178,E2 -19282.178} C_VEL
LIN {X 0,Y 242.067,Z 289.955,A -85,B 0,C 180,E1 -19285.836,E2 -19285.836} C_VEL
LIN {X 0,Y 242.007,Z 289.955,A -85,B 0,C 180,E1 -19289.581,E2 -19289.581} C_VEL
LIN {X 0,Y 241.99,Z 289.965,A -85,B 0,C 180,E1 -19293.488,E2 -19293.488} C_VEL
LIN {X 0,Y 242.002,Z 289.959,A -85,B 0,C 180,E1 -19297.577,E2 -19297.577} C_VEL
LIN {X 0,Y 241.953,Z 289.961,A -85,B 0,C 180,E1 -19301.916,E2 -19301.916} C_VEL
LIN {X 0,Y 241.988,Z 289.966,A -85,B 0,C 180,E1 -19306.555,E2 -19306.555} C_VEL
LIN {X 0,Y 242.004,Z 289.959,A -85,B 0,C 180,E1 -19310.289,E2 -19310.289} C_VEL
LIN {X 0,Y 242.032,Z 289.953,A -85,B 0,C 180,E1 -19314.495,E2 -19314.495} C_VEL
LIN {X 0,Y 241.971,Z 289.969,A -85,B 0,C 180,E1 -19318.478,E2 -19318.478} C_VEL
LIN {X 0,Y 242.006,Z 289.967,A -85,B 0,C 180,E1 -19322.311,E2 -19322.311} C_VEL
LIN {X 0,Y 242.051,Z 289.961,A -85,B 0,C 180,E1 -19326.014,E2 -19326.014} C_VEL
LIN {X 0,Y 242.03,Z 289.96,A -85,B 0,C 180,E1 -19329.606,E2 -19329.606} C_VEL
LIN {X 0,Y 242.156,Z 289.943,A -85,B 0,C 180,E1 -19333.277,E2 -19333.277} C_VEL
LIN {X 0,Y 242.178,Z 289.94,A -85,B 0,C 180,E1 -19338.278,E2 -19338.278} C_VEL
LIN {X 0,Y 242.372,Z 289.918,A -85,B 0,C 180,E1 -19340.56,E2 -19340.56} C_VEL
LIN {X 0,Y 243.42,Z 292.797,A -85,B 0,C 180,E1 -19340.914,E2 -19340.914} C_VEL
LIN {X 0,Y 245.075,Z 295.131,A -85,B 0,C 180,E1 -19341.325,E2 -19341.325} C_VEL
LIN {X 0,Y 250.359,Z 305.052,A -85,B 0,C 180,E1 -19342.868,E2 -19342.868} C_VEL
LIN {X 0,Y 255.877,Z 316.577,A -85,B 0,C 180,E1 -19344.669,E2 -19344.669} C_VEL
LIN {X 0,Y 259.75,Z 329.598,A -85,B 0,C 180,E1 -19346.535,E2 -19346.535} C_VEL
LIN {X 0,Y 262.692,Z 340.064,A -85,B 0,C 180,E1 -19348.182,E2 -19348.182} C_VEL
LIN {X 0,Y 264.235,Z 347.42,A -85,B 0,C 180,E1 -19349.37,E2 -19349.37} C_VEL
LIN {X 0,Y 261.659,Z 360.055,A -85,B 0,C 180,E1 -19350.961,E2 -19350.961} C_VEL
LIN {X 0,Y 258.431,Z 373.003,A -85,B 0,C 180,E1 -19352.938,E2 -19352.938} C_VEL
LIN {X 0,Y 255.445,Z 384.279,A -85,B 0,C 180,E1 -19355.049,E2 -19355.049} C_VEL
LIN {X 0,Y 252.188,Z 395.495,A -85,B 0,C 180,E1 -19357.606,E2 -19357.606} C_VEL
LIN {X 0,Y 249.458,Z 404.514,A -85,B 0,C 180,E1 -19360.099,E2 -19360.099} C_VEL
LIN {X 0,Y 246.624,Z 413.603,A -85,B 0,C 180,E1 -19363.177,E2 -19363.177} C_VEL
LIN {X 0,Y 244.725,Z 419.946,A -85,B 0,C 180,E1 -19365.831,E2 -19365.831} C_VEL
LIN {X 0,Y 243.093,Z 425.323,A -85,B 0,C 180,E1 -19368.542,E2 -19368.542} C_VEL
LIN {X 0,Y 241.836,Z 430.156,A -85,B 0,C 180,E1 -19371.58,E2 -19371.58} C_VEL
LIN {X 0,Y 240.734,Z 434.409,A -85,B 0,C 180,E1 -19375.18,E2 -19375.18} C_VEL
LIN {X 0,Y 240.1,Z 437.127,A -85,B 0,C 180,E1 -19378.587,E2 -19378.587} C_VEL
LIN {X 0,Y 239.869,Z 438.559,A -85,B 0,C 180,E1 -19381.828,E2 -19381.828} C_VEL
LIN {X 0,Y 239.921,Z 438.968,A -85,B 0,C 180,E1 -19384.899,E2 -19384.899} C_VEL
LIN {X 0,Y 240.234,Z 438.496,A -85,B 0,C 180,E1 -19387.903,E2 -19387.903} C_VEL
LIN {X 0,Y 240.835,Z 437.204,A -85,B 0,C 180,E1 -19390.652,E2 -19390.652} C_VEL
LIN {X 0,Y 242.022,Z 434.444,A -85,B 0,C 180,E1 -19394.179,E2 -19394.179} C_VEL
LIN {X 0,Y 243.591,Z 430.785,A -85,B 0,C 180,E1 -19397.366,E2 -19397.366} C_VEL
LIN {X 0,Y 246.073,Z 424.898,A -85,B 0,C 180,E1 -19401.076,E2 -19401.076} C_VEL
LIN {X 0,Y 248.668,Z 418.71,A -85,B 0,C 180,E1 -19404.081,E2 -19404.081} C_VEL
LIN {X 0,Y 251.7,Z 411.473,A -85,B 0,C 180,E1 -19406.892,E2 -19406.892} C_VEL
LIN {X 0,Y 254.965,Z 403.325,A -85,B 0,C 180,E1 -19409.471,E2 -19409.471} C_VEL
LIN {X 0,Y 258.698,Z 393.601,A -85,B 0,C 180,E1 -19411.994,E2 -19411.994} C_VEL
LIN {X 0,Y 262.415,Z 383.425,A -85,B 0,C 180,E1 -19414.145,E2 -19414.145} C_VEL
LIN {X 0,Y 266.058,Z 372.215,A -85,B 0,C 180,E1 -19416.116,E2 -19416.116} C_VEL
LIN {X 0,Y 269.871,Z 359.217,A -85,B 0,C 180,E1 -19417.979,E2 -19417.979} C_VEL
LIN {X 0,Y 270.901,Z 355.143,A -85,B 0,C 180,E1 -19418.505,E2 -19418.505} C_VEL
LIN {X 0,Y 269.016,Z 344.815,A -85,B 0,C 180,E1 -19420.545,E2 -19420.545} C_VEL
LIN {X 0,Y 266.043,Z 334.316,A -85,B 0,C 180,E1 -19422.712,E2 -19422.712} C_VEL
LIN {X 0,Y 261.784,Z 323.537,A -85,B 0,C 180,E1 -19425.117,E2 -19425.117} C_VEL
LIN {X 0,Y 257.419,Z 315.169,A -85,B 0,C 180,E1 -19427.254,E2 -19427.254} C_VEL
LIN {X 0,Y 255.654,Z 312.2,A -85,B 0,C 180,E1 -19428.077,E2 -19428.077} C_VEL
